KUKA KRL program: MyProgram_024().src

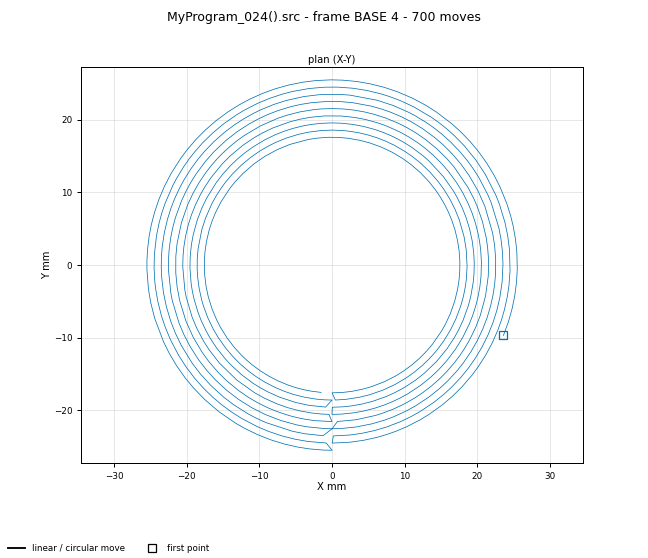
[picture p0: tool path of MyProgram_024().src in frame BASE 4, 700 of 700 moves have a stored position in this frame; points joined in program order, loops and branches not executed]
&ACCESS RVP
&REL 1
&PARAM TEMPLATE = C:\KRC\Roboter\Template\vorgabe
&PARAM EDITMASK = *
DEF MyProgram_024()
; ---- Setting reference (Base) ----
$BASE = BASE_DATA[4]

; --------------------------
; ---- Setting tool (TCP) ----
$TOOL = TOOL_DATA[3]
; --------------------------

$VEL.CP = VEL_APROX_PRINT
Startdeposition()
$VEL.CP = VEL_PRINT
LIN {X 23.5974,Y -9.6926,Z 57,A -28.3314,B 24.8282,C -3.0231,E1 25.1491,E2 -248.9797} C_DIS
LIN {X 24.2747,Y -7.8424,Z 57,A -24.218,B 24.8271,C -3.0328,E1 25.1528,E2 -253.093} C_DIS
LIN {X 24.7886,Y -6.0243,Z 57,A -19.8606,B 24.8255,C -3.0472,E1 25.1559,E2 -257.4593} C_DIS
LIN {X 25.1579,Y -4.2259,Z 57,A -15.7449,B 24.824,C -3.0599,E1 25.158,E2 -261.5811} C_DIS
LIN {X 25.4033,Y -2.3332,Z 57,A -11.6875,B 24.8228,C -3.0706,E1 25.1593,E2 -265.6398} C_DIS
LIN {X 25.5049,Y -0.5316,Z 57,A -6.9801,B 24.8204,C -3.0909,E1 25.1598,E2 -270.3674} C_DIS
LIN {X 25.4452,Y 1.817,Z 57,A -2.3084,B 24.8193,C -3.1002,E1 25.1592,E2 -275.0333} C_DIS
LIN {X 25.2568,Y 3.5873,Z 57,A 1.7378,B 24.8178,C -3.113,E1 25.1578,E2 -279.0859} C_DIS
LIN {X 24.9227,Y 5.4431,Z 57,A 5.9882,B 24.8163,C -3.1259,E1 25.1554,E2 -283.3422} C_DIS
LIN {X 24.5979,Y 6.7615,Z 57,A 9.2535,B 24.8149,C -3.1375,E1 25.1531,E2 -286.6161} C_DIS
LIN {X 24.0961,Y 8.3747,Z 57,A 13.4975,B 24.813,C -3.1536,E1 25.1492,E2 -290.8744} C_DIS
LIN {X 23.1444,Y 10.7284,Z 57,A 18.4456,B 24.8121,C -3.1608,E1 25.1437,E2 -295.8124} C_DIS
LIN {X 22.2888,Y 12.4091,Z 57,A 22.6691,B 24.8108,C -3.1719,E1 25.1382,E2 -300.0401} C_DIS
LIN {X 21.2717,Y 14.0817,Z 57,A 27.0653,B 24.8095,C -3.1829,E1 25.1316,E2 -304.4403} C_DIS
LIN {X 20.123,Y 15.6796,Z 57,A 31.2435,B 24.8085,C -3.1908,E1 25.1246,E2 -308.6172} C_DIS
LIN {X 19.0448,Y 16.9728,Z 57,A 35.1391,B 24.8074,C -3.2004,E1 25.1175,E2 -312.518} C_DIS
LIN {X 17.7974,Y 18.2769,Z 57,A 39.241,B 24.8063,C -3.2093,E1 25.1094,E2 -316.6237} C_DIS
LIN {X 16.5553,Y 19.4087,Z 57,A 43.3186,B 24.805,C -3.2197,E1 25.1008,E2 -320.7097} C_DIS
LIN {X 14.3642,Y 21.082,Z 57,A 49.1701,B 24.8042,C -3.2265,E1 25.0876,E2 -326.5568} C_DIS
LIN {X 12.7921,Y 22.0714,Z 57,A 53.3227,B 24.8035,C -3.2324,E1 25.0777,E2 -330.7103} C_DIS
LIN {X 11.0794,Y 22.9786,Z 57,A 57.9272,B 24.8025,C -3.2401,E1 25.0662,E2 -335.3208} C_DIS
LIN {X 9.0363,Y 23.856,Z 57,A 62.7399,B 24.8021,C -3.2433,E1 25.0537,E2 -340.1302} C_DIS
LIN {X 7.1477,Y 24.4882,Z 57,A 67.1046,B 24.8019,C -3.2456,E1 25.0421,E2 -344.4925} C_DIS
LIN {X 5.2619,Y 24.9618,Z 57,A 71.4856,B 24.8016,C -3.248,E1 25.0302,E2 -348.873} C_DIS
LIN {X 3.3906,Y 25.284,Z 57,A 75.7755,B 24.8014,C -3.2494,E1 25.0184,E2 -353.1622} C_DIS
LIN {X 1.4533,Y 25.4688,Z 57,A 79.6015,B 24.8019,C -3.245,E1 25.0077,E2 -356.9757} C_DIS
LIN {X -0.1497,Y 25.5099,Z 57,A 83.8568,B 24.8013,C -3.2498,E1 24.9958,E2 -361.2422} C_DIS
LIN {X -2.166,Y 25.4178,Z 57,A 88.1783,B 24.8018,C -3.2463,E1 24.9838,E2 -365.5568} C_DIS
LIN {X -3.9428,Y 25.2038,Z 57,A 92.4799,B 24.8018,C -3.246,E1 24.9719,E2 -369.8611} C_DIS
LIN {X -5.9691,Y 24.8019,Z 57,A 96.9208,B 24.8025,C -3.2405,E1 24.9598,E2 -374.2945} C_DIS
LIN {X -7.8398,Y 24.2755,Z 57,A 101.2468,B 24.8031,C -3.2355,E1 24.9483,E2 -378.6158} C_DIS
LIN {X -9.6059,Y 23.6324,Z 57,A 105.5538,B 24.8037,C -3.2306,E1 24.9371,E2 -382.9204} C_DIS
LIN {X -11.3897,Y 22.8266,Z 57,A 109.6739,B 24.8047,C -3.2221,E1 24.9267,E2 -387.0305} C_DIS
LIN {X -12.8693,Y 22.0267,Z 57,A 113.4295,B 24.8055,C -3.2156,E1 24.9175,E2 -390.7813} C_DIS
LIN {X -14.3968,Y 21.0597,Z 57,A 117.8771,B 24.8061,C -3.2105,E1 24.9072,E2 -395.2315} C_DIS
LIN {X -15.9987,Y 19.8702,Z 57,A 122.312,B 24.8073,C -3.201,E1 24.8974,E2 -399.6598} C_DIS
LIN {X -17.4613,Y 18.5978,Z 57,A 126.6023,B 24.8085,C -3.1909,E1 24.8885,E2 -403.9432} C_DIS
LIN {X -18.7226,Y 17.3277,Z 57,A 130.7535,B 24.8096,C -3.1821,E1 24.8805,E2 -408.0912} C_DIS
LIN {X -19.9337,Y 15.9198,Z 57,A 134.7937,B 24.8109,C -3.1708,E1 24.8733,E2 -412.1231} C_DIS
LIN {X -20.8288,Y 14.7286,Z 57,A 138.4822,B 24.8117,C -3.164,E1 24.8673,E2 -415.8132} C_DIS
LIN {X -22.187,Y 12.5909,Z 57,A 144.0705,B 24.8137,C -3.1477,E1 24.8592,E2 -421.3912} C_DIS
LIN {X -23.0971,Y 10.8307,Z 57,A 148.4759,B 24.8152,C -3.1346,E1 24.8538,E2 -425.789} C_DIS
LIN {X -23.8551,Y 9.0389,Z 57,A 152.9416,B 24.8167,C -3.1222,E1 24.8491,E2 -430.25} C_DIS
LIN {X -24.4663,Y 7.2223,Z 57,A 157.3061,B 24.8182,C -3.1095,E1 24.8455,E2 -434.609} C_DIS
LIN {X -24.9012,Y 5.5426,Z 57,A 160.8222,B 24.8199,C -3.0955,E1 24.8432,E2 -438.1121} C_DIS
LIN {X -25.2019,Y 3.9555,Z 57,A 164.8469,B 24.8209,C -3.0864,E1 24.8413,E2 -442.1389} C_DIS
LIN {X -25.4178,Y 2.1663,Z 57,A 168.8418,B 24.8224,C -3.0735,E1 24.8401,E2 -446.1268} C_DIS
LIN {X -25.5037,Y 0.5661,Z 57,A 171.8056,B 24.8241,C -3.0589,E1 24.8398,E2 -449.0735} C_DIS
LIN {X -25.5018,Y -0.6552,Z 57,A 175.5636,B 24.8245,C -3.0558,E1 24.84,E2 -452.8467} C_DIS
LIN {X -25.2925,Y -3.3258,Z 57,A -178.4748,B 24.8266,C -3.037,E1 24.8416,E2 -458.7989} C_DIS
LIN {X -24.9832,Y -5.1588,Z 57,A -174.3635,B 24.8281,C -3.024,E1 24.8438,E2 -462.9035} C_DIS
LIN {X -24.4374,Y -7.3208,Z 57,A -168.6261,B 24.8293,C -3.0134,E1 24.8481,E2 -468.6488} C_DIS
LIN {X -23.2088,Y -10.5894,Z 57,A -161.9405,B 24.8326,C -2.9847,E1 24.855,E2 -475.3029} C_DIS
LIN {X -22.4165,Y -12.1769,Z 57,A -157.4517,B 24.8334,C -2.977,E1 24.8608,E2 -479.7974} C_DIS
LIN {X -21.4191,Y -13.8564,Z 57,A -153.0174,B 24.8347,C -2.9662,E1 24.8673,E2 -484.2283} C_DIS
LIN {X -20.2689,Y -15.4905,Z 57,A -148.5031,B 24.8358,C -2.9557,E1 24.8748,E2 -488.7393} C_DIS
LIN {X -19.0968,Y -16.9142,Z 57,A -144.3818,B 24.8369,C -2.9463,E1 24.8823,E2 -492.857} C_DIS
LIN {X -17.5052,Y -18.5563,Z 57,A -138.9873,B 24.8378,C -2.9376,E1 24.893,E2 -498.2534} C_DIS
LIN {X -15.5207,Y -20.2452,Z 57,A -132.526,B 24.8385,C -2.9313,E1 24.9071,E2 -504.724} C_DIS
LIN {X -13.3044,Y -21.7661,Z 57,A -127.5351,B 24.8404,C -2.9147,E1 24.9187,E2 -509.6914} C_DIS
LIN {X -12.0506,Y -22.4847,Z 57,A -123.9663,B 24.8406,C -2.9128,E1 24.9274,E2 -513.2659} C_DIS
LIN {X -10.2372,Y -23.3661,Z 57,A -119.449,B 24.8411,C -2.9078,E1 24.9389,E2 -517.7823} C_DIS
LIN {X -8.4417,Y -24.0728,Z 57,A -115.0933,B 24.8415,C -2.9042,E1 24.9503,E2 -522.1384} C_DIS
LIN {X -6.6102,Y -24.6387,Z 57,A -110.8019,B 24.8418,C -2.9013,E1 24.9618,E2 -526.4299} C_DIS
LIN {X -4.7543,Y -25.0634,Z 57,A -106.5325,B 24.842,C -2.8994,E1 24.9735,E2 -530.6999} C_DIS
LIN {X -3.1602,Y -25.314,Z 57,A -102.8759,B 24.842,C -2.899,E1 24.9836,E2 -534.3583} C_DIS
LIN {X -1.1779,Y -25.483,Z 57,A -98.4765,B 24.8421,C -2.8985,E1 24.9958,E2 -538.758} C_DIS
LIN {X 0.0017,Y -25.5054,Z 57,A -95.9196,B 24.8421,C -2.8983,E1 25.003,E2 -541.3145} C_DIS
Enddeposition()
LIN {X 0.0017,Y -25.5054,Z 57,A -95.9196,B 24.8421,C -2.8983,E1 25.003,E2 -541.3145} C_DIS
Startdeposition()
$VEL.CP = VEL_PRINT
LIN {X -0.8162,Y -24.5086,Z 57,A -100.4797,B 24.8428,C -2.8929,E1 24.9902,E2 -536.7411} C_DIS
LIN {X -3.343,Y -24.2934,Z 57,A -105.8436,B 24.8422,C -2.898,E1 24.9753,E2 -531.386} C_DIS
LIN {X -5.1134,Y -23.9829,Z 57,A -110.0123,B 24.842,C -2.8998,E1 24.9639,E2 -527.217} C_DIS
LIN {X -6.9312,Y -23.5218,Z 57,A -114.4025,B 24.8417,C -2.9024,E1 24.9521,E2 -522.8262} C_DIS
LIN {X -8.7143,Y -22.9213,Z 57,A -118.9495,B 24.8414,C -2.905,E1 24.9401,E2 -518.2763} C_DIS
LIN {X -10.284,Y -22.2612,Z 57,A -123.2424,B 24.8412,C -2.9071,E1 24.9292,E2 -513.978} C_DIS
LIN {X -12.5044,Y -21.0944,Z 57,A -128.2625,B 24.8397,C -2.9204,E1 24.917,E2 -508.9752} C_DIS
LIN {X -13.8365,Y -20.2452,Z 57,A -132.1033,B 24.8392,C -2.925,E1 24.908,E2 -505.133} C_DIS
LIN {X -15.1839,Y -19.2557,Z 57,A -136.3359,B 24.8387,C -2.9296,E1 24.8986,E2 -500.8961} C_DIS
LIN {X -16.5203,Y -18.1223,Z 57,A -140.2889,B 24.8378,C -2.9382,E1 24.8903,E2 -496.9481} C_DIS
LIN {X -17.6802,Y -16.9922,Z 57,A -144.3432,B 24.8371,C -2.9444,E1 24.8823,E2 -492.8914} C_DIS
LIN {X -18.9103,Y -15.6122,Z 57,A -148.5343,B 24.8359,C -2.9548,E1 24.8747,E2 -488.7059} C_DIS
LIN {X -20.0676,Y -14.0935,Z 57,A -153.0925,B 24.8348,C -2.9648,E1 24.8672,E2 -484.1497} C_DIS
LIN {X -21.1149,Y -12.4698,Z 57,A -158.0469,B 24.8338,C -2.974,E1 24.86,E2 -479.1918} C_DIS
LIN {X -22.2501,Y -10.3079,Z 57,A -162.6904,B 24.8314,C -2.9949,E1 24.8542,E2 -474.5733} C_DIS
LIN {X -22.9755,Y -8.5693,Z 57,A -167.9487,B 24.8305,C -3.0028,E1 24.8487,E2 -469.3047} C_DIS
LIN {X -23.5095,Y -6.9732,Z 57,A -171.3197,B 24.8289,C -3.0171,E1 24.8459,E2 -465.9484} C_DIS
LIN {X -24.0022,Y -5.0236,Z 57,A -177.0526,B 24.8279,C -3.026,E1 24.8423,E2 -460.2034} C_DIS
LIN {X -24.3161,Y -3.1693,Z 57,A 179.493,B 24.8258,C -3.044,E1 24.8409,E2 -456.7713} C_DIS
LIN {X -24.4335,Y -2.0783,Z 57,A 176.5746,B 24.8251,C -3.0501,E1 24.8401,E2 -453.8502} C_DIS
LIN {X -24.5179,Y -0.4555,Z 57,A 172.7447,B 24.8238,C -3.0618,E1 24.8398,E2 -450.0252} C_DIS
LIN {X -24.4799,Y 1.4247,Z 57,A 168.2785,B 24.8222,C -3.0751,E1 24.8403,E2 -445.5641} C_DIS
LIN {X -24.1837,Y 4.0593,Z 57,A 161.6445,B 24.8202,C -3.0923,E1 24.8427,E2 -438.9316} C_DIS
LIN {X -23.8193,Y 5.828,Z 57,A 158.2213,B 24.8183,C -3.1091,E1 24.8448,E2 -435.5285} C_DIS
LIN {X -23.4594,Y 7.1394,Z 57,A 154.6095,B 24.8174,C -3.1167,E1 24.8476,E2 -431.914} C_DIS
LIN {X -23.0092,Y 8.4797,Z 57,A 150.6203,B 24.8166,C -3.1233,E1 24.8514,E2 -427.918} C_DIS
LIN {X -21.9422,Y 10.9487,Z 57,A 145.374,B 24.8138,C -3.1467,E1 24.8575,E2 -422.6991} C_DIS
LIN {X -21.429,Y 11.9218,Z 57,A 142.3229,B 24.8132,C -3.1515,E1 24.8616,E2 -419.6435} C_DIS
LIN {X -20.4509,Y 13.5307,Z 57,A 138.2469,B 24.8116,C -3.1652,E1 24.8676,E2 -415.5796} C_DIS
LIN {X -19.6571,Y 14.6605,Z 57,A 135.1759,B 24.8105,C -3.1745,E1 24.8726,E2 -412.516} C_DIS
LIN {X -18.9586,Y 15.5535,Z 57,A 132.147,B 24.8099,C -3.1793,E1 24.8779,E2 -409.4842} C_DIS
LIN {X -17.8107,Y 16.8557,Z 57,A 127.8837,B 24.8089,C -3.188,E1 24.886,E2 -405.2229} C_DIS
LIN {X -16.3984,Y 18.2327,Z 57,A 123.2379,B 24.8076,C -3.1982,E1 24.8954,E2 -400.5827} C_DIS
LIN {X -14.9317,Y 19.4519,Z 57,A 118.4259,B 24.8068,C -3.2055,E1 24.9059,E2 -395.7702} C_DIS
LIN {X -13.2236,Y 20.6511,Z 57,A 114.2463,B 24.8051,C -3.2189,E1 24.9156,E2 -391.6087} C_DIS
LIN {X -12.1128,Y 21.3219,Z 57,A 110.8599,B 24.8048,C -3.222,E1 24.9237,E2 -388.2195} C_DIS
LIN {X -10.3297,Y 22.24,Z 57,A 106.1341,B 24.8039,C -3.229,E1 24.9356,E2 -383.498} C_DIS
LIN {X -8.5761,Y 22.9732,Z 57,A 101.6704,B 24.8032,C -3.2347,E1 24.9472,E2 -379.0384} C_DIS
LIN {X -6.7424,Y 23.5769,Z 57,A 97.607,B 24.8022,C -3.2427,E1 24.958,E2 -374.9871} C_DIS
LIN {X -5.4397,Y 23.9109,Z 57,A 93.8987,B 24.8023,C -3.2417,E1 24.968,E2 -371.2712} C_DIS
LIN {X -3.1801,Y 24.3149,Z 57,A 88.636,B 24.8018,C -3.246,E1 24.9825,E2 -366.0141} C_DIS
LIN {X -1.0603,Y 24.4985,Z 57,A 83.951,B 24.8013,C -3.2502,E1 24.9956,E2 -361.3373} C_DIS
LIN {X 0.7326,Y 24.5108,Z 57,A 79.1328,B 24.8018,C -3.246,E1 25.009,E2 -356.5096} C_DIS
LIN {X 2.8302,Y 24.3581,Z 57,A 74.5816,B 24.8015,C -3.2484,E1 25.0217,E2 -351.9668} C_DIS
LIN {X 4.7024,Y 24.067,Z 57,A 69.4413,B 24.8024,C -3.2409,E1 25.0358,E2 -346.8144} C_DIS
LIN {X 6.6864,Y 23.5927,Z 57,A 65.7695,B 24.8017,C -3.2473,E1 25.0457,E2 -343.1636} C_DIS
LIN {X 7.8457,Y 23.2327,Z 57,A 62.9862,B 24.8019,C -3.2456,E1 25.0531,E2 -340.3814} C_DIS
LIN {X 9.3946,Y 22.6509,Z 57,A 58.3374,B 24.8032,C -3.2349,E1 25.0652,E2 -335.7176} C_DIS
LIN {X 11.2204,Y 21.8043,Z 57,A 53.3946,B 24.8041,C -3.2271,E1 25.0775,E2 -330.7694} C_DIS
LIN {X 13.6548,Y 20.3686,Z 57,A 47.7894,B 24.8041,C -3.2267,E1 25.0908,E2 -325.1811} C_DIS
LIN {X 14.7224,Y 19.6108,Z 57,A 44.6371,B 24.8049,C -3.2207,E1 25.0979,E2 -322.0257} C_DIS
LIN {X 15.8085,Y 18.7463,Z 57,A 41.3255,B 24.8057,C -3.2141,E1 25.1051,E2 -318.7111} C_DIS
LIN {X 16.8223,Y 17.8422,Z 57,A 37.9278,B 24.8067,C -3.2056,E1 25.1121,E2 -315.3071} C_DIS
LIN {X 18.1912,Y 16.4443,Z 57,A 33.2587,B 24.808,C -3.1949,E1 25.121,E2 -310.6329} C_DIS
LIN {X 19.8061,Y 14.4585,Z 57,A 26.7554,B 24.8104,C -3.1756,E1 25.1321,E2 -304.1145} C_DIS
LIN {X 21.0994,Y 12.4958,Z 57,A 21.1531,B 24.8122,C -3.1604,E1 25.1403,E2 -298.5048} C_DIS
LIN {X 22.5618,Y 9.6075,Z 57,A 15.2266,B 24.8125,C -3.1574,E1 25.1474,E2 -292.6028} C_DIS
LIN {X 23.0349,Y 8.4095,Z 57,A 11.0682,B 24.815,C -3.1364,E1 25.1515,E2 -288.4179} C_DIS
LIN {X 23.8129,Y 5.8544,Z 57,A 5.2905,B 24.8166,C -3.123,E1 25.1559,E2 -282.6417} C_DIS
LIN {X 24.1913,Y 4.0145,Z 57,A 0.9918,B 24.8181,C -3.1108,E1 25.1581,E2 -278.339} C_DIS
LIN {X 24.4273,Y 2.1521,Z 57,A -4.0505,B 24.8205,C -3.09,E1 25.1595,E2 -273.2775} C_DIS
LIN {X 24.5108,Y -0.7385,Z 57,A -10.2973,B 24.8223,C -3.0746,E1 25.1595,E2 -267.0314} C_DIS
LIN {X 24.3597,Y -2.8172,Z 57,A -14.5236,B 24.8232,C -3.0666,E1 25.1585,E2 -262.8111} C_DIS
LIN {X 24.1391,Y -4.317,Z 57,A -18.4922,B 24.825,C -3.0508,E1 25.1567,E2 -258.8285} C_DIS
LIN {X 23.7335,Y -6.1692,Z 57,A -22.9517,B 24.8266,C -3.0368,E1 25.1538,E2 -254.3617} C_DIS
LIN {X 23.2874,Y -7.6821,Z 57,A -26.0063,B 24.8271,C -3.0326,E1 25.1513,E2 -251.3144} C_DIS
LIN {X 22.8272,Y -8.9576,Z 57,A -29.674,B 24.8288,C -3.0176,E1 25.1477,E2 -247.6317} C_DIS
LIN {X 22.0848,Y -10.6578,Z 57,A -33.9482,B 24.8302,C -3.0056,E1 25.1427,E2 -243.3521} C_DIS
LIN {X 21.2084,Y -12.3104,Z 57,A -38.7058,B 24.8321,C -2.9891,E1 25.1362,E2 -238.5801} C_DIS
LIN {X 20.088,Y -14.0645,Z 57,A -42.8035,B 24.8326,C -2.9841,E1 25.1299,E2 -234.4909} C_DIS
LIN {X 19.2809,Y -15.152,Z 57,A -46.285,B 24.834,C -2.9724,E1 25.1239,E2 -230.9983} C_DIS
LIN {X 17.9089,Y -16.7511,Z 57,A -51.0916,B 24.8352,C -2.9614,E1 25.115,E2 -226.1872} C_DIS
LIN {X 16.5964,Y -18.0525,Z 57,A -55.5524,B 24.8365,C -2.95,E1 25.106,E2 -221.7177} C_DIS
LIN {X 15.203,Y -19.2406,Z 57,A -60.0611,B 24.8377,C -2.9385,E1 25.0962,E2 -217.1988} C_DIS
LIN {X 13.3435,Y -20.5736,Z 57,A -64.6446,B 24.8381,C -2.9356,E1 25.0857,E2 -212.6241} C_DIS
LIN {X 12.0817,Y -21.3389,Z 57,A -68.6968,B 24.8394,C -2.9236,E1 25.0759,E2 -208.5558} C_DIS
LIN {X 10.2776,Y -22.2641,Z 57,A -73.2647,B 24.84,C -2.9178,E1 25.0644,E2 -203.9862} C_DIS
LIN {X 8.8215,Y -22.8801,Z 57,A -76.4646,B 24.84,C -2.9173,E1 25.0562,E2 -200.7925} C_DIS
LIN {X 7.6695,Y -23.2913,Z 57,A -79.7044,B 24.8408,C -2.9103,E1 25.0476,E2 -197.5423} C_DIS
LIN {X 6.2074,Y -23.7233,Z 57,A -83.3054,B 24.8413,C -2.9062,E1 25.0379,E2 -193.9375} C_DIS
LIN {X 4.3572,Y -24.1319,Z 57,A -87.7631,B 24.8417,C -2.9022,E1 25.0257,E2 -189.4757} C_DIS
LIN {X 2.4426,Y -24.4001,Z 57,A -92.708,B 24.8424,C -2.8959,E1 25.0119,E2 -184.5194} C_DIS
LIN {X 0.0065,Y -24.5225,Z 57,A -95.59,B 24.84,C -2.9177,E1 25.004,E2 -181.6903} C_DIS
Enddeposition()
LIN {X 0.0065,Y -24.5225,Z 57,A -95.59,B 24.84,C -2.9177,E1 25.004,E2 -181.6903} C_DIS
Startdeposition()
$VEL.CP = VEL_PRINT
LIN {X 0.1728,Y -23.5332,Z 57,A -95.0814,B 24.8381,C -2.9354,E1 25.0056,E2 -182.241} C_DIS
LIN {X 2.4377,Y -23.4068,Z 57,A -90.2543,B 24.8384,C -2.9321,E1 25.019,E2 -187.0578} C_DIS
LIN {X 4.046,Y -23.1837,Z 57,A -85.8902,B 24.8377,C -2.9385,E1 25.031,E2 -191.4327} C_DIS
LIN {X 5.8549,Y -22.7937,Z 57,A -81.6004,B 24.8375,C -2.9408,E1 25.0427,E2 -195.722} C_DIS
LIN {X 7.5378,Y -22.2935,Z 57,A -76.8383,B 24.8364,C -2.9502,E1 25.0554,E2 -200.4977} C_DIS
LIN {X 9.3798,Y -21.5835,Z 57,A -72.4094,B 24.8361,C -2.9534,E1 25.0668,E2 -204.9239} C_DIS
LIN {X 10.8597,Y -20.8786,Z 57,A -68.6996,B 24.8357,C -2.9571,E1 25.0761,E2 -208.6324} C_DIS
LIN {X 12.1662,Y -20.1452,Z 57,A -64.7539,B 24.8346,C -2.9664,E1 25.0856,E2 -212.5883} C_DIS
LIN {X 14.0298,Y -18.8948,Z 57,A -59.3169,B 24.8334,C -2.9769,E1 25.0981,E2 -218.0315} C_DIS
LIN {X 15.404,Y -17.7921,Z 57,A -55.2869,B 24.8327,C -2.9836,E1 25.1067,E2 -222.0618} C_DIS
LIN {X 16.512,Y -16.7688,Z 57,A -51.5293,B 24.8316,C -2.993,E1 25.1143,E2 -225.8261} C_DIS
LIN {X 17.7863,Y -15.411,Z 57,A -47.3126,B 24.8308,C -3.0008,E1 25.1222,E2 -230.0428} C_DIS
LIN {X 18.8448,Y -14.0963,Z 57,A -42.8149,B 24.8291,C -3.0156,E1 25.13,E2 -234.5542} C_DIS
LIN {X 19.7762,Y -12.757,Z 57,A -39.0539,B 24.8281,C -3.0241,E1 25.1358,E2 -238.3168} C_DIS
LIN {X 20.6346,Y -11.3168,Z 57,A -34.7573,B 24.8265,C -3.0379,E1 25.1418,E2 -242.6239} C_DIS
LIN {X 21.4569,Y -9.666,Z 57,A -30.3654,B 24.8251,C -3.0499,E1 25.147,E2 -247.0205} C_DIS
LIN {X 22.1456,Y -7.9621,Z 57,A -25.9982,B 24.8237,C -3.0621,E1 25.1514,E2 -251.3923} C_DIS
LIN {X 22.6902,Y -6.2446,Z 57,A -21.4937,B 24.822,C -3.0768,E1 25.1549,E2 -255.9059} C_DIS
LIN {X 23.0932,Y -4.5333,Z 57,A -17.297,B 24.8206,C -3.0891,E1 25.1574,E2 -260.1073} C_DIS
LIN {X 23.4185,Y -2.3263,Z 57,A -11.3589,B 24.818,C -3.1117,E1 25.1594,E2 -266.0637} C_DIS
LIN {X 23.5357,Y 0.142,Z 57,A -5.7796,B 24.8163,C -3.1255,E1 25.1597,E2 -271.6427} C_DIS
LIN {X 23.461,Y 1.8498,Z 57,A -2.1065,B 24.8154,C -3.1331,E1 25.1591,E2 -275.3119} C_DIS
LIN {X 23.2709,Y 3.509,Z 57,A 2.26,B 24.8136,C -3.1488,E1 25.1575,E2 -279.6899} C_DIS
LIN {X 22.9699,Y 5.1217,Z 57,A 7.3044,B 24.8108,C -3.1723,E1 25.1545,E2 -284.7608} C_DIS
LIN {X 21.9227,Y 8.557,Z 57,A 14.7705,B 24.8094,C -3.1836,E1 25.1478,E2 -292.2114} C_DIS
LIN {X 21.4484,Y 9.6849,Z 57,A 18.4083,B 24.8076,C -3.1989,E1 25.1437,E2 -295.8657} C_DIS
LIN {X 20.1752,Y 12.1166,Z 57,A 24.0792,B 24.8067,C -3.2057,E1 25.136,E2 -301.5232} C_DIS
LIN {X 19.342,Y 13.4062,Z 57,A 27.7241,B 24.8057,C -3.2141,E1 25.1304,E2 -305.1698} C_DIS
LIN {X 18.6123,Y 14.4023,Z 57,A 30.9154,B 24.8046,C -3.2231,E1 25.125,E2 -308.3672} C_DIS
LIN {X 17.7311,Y 15.4742,Z 57,A 34.6473,B 24.8033,C -3.2342,E1 25.1183,E2 -312.1085} C_DIS
LIN {X 16.411,Y 16.8681,Z 57,A 39.2881,B 24.8021,C -3.2436,E1 25.1091,E2 -316.7517} C_DIS
LIN {X 15.0831,Y 18.0649,Z 57,A 43.2663,B 24.8016,C -3.2481,E1 25.1008,E2 -320.7252} C_DIS
LIN {X 13.9703,Y 18.9386,Z 57,A 46.6692,B 24.8009,C -3.2537,E1 25.0932,E2 -324.1289} C_DIS
LIN {X 12.9444,Y 19.6541,Z 57,A 49.9429,B 24.8,C -3.2607,E1 25.0856,E2 -327.4081} C_DIS
LIN {X 11.4624,Y 20.5535,Z 57,A 53.7393,B 24.7998,C -3.2627,E1 25.0765,E2 -331.1978} C_DIS
LIN {X 10.4876,Y 21.0677,Z 57,A 56.7363,B 24.799,C -3.2688,E1 25.069,E2 -334.2013} C_DIS
LIN {X 8.401,Y 21.9831,Z 57,A 63.2209,B 24.7973,C -3.2827,E1 25.0522,E2 -340.7039} C_DIS
LIN {X 6.1651,Y 22.7118,Z 57,A 69.2316,B 24.7965,C -3.289,E1 25.0361,E2 -346.7194} C_DIS
LIN {X 2.4387,Y 23.407,Z 57,A 76.8785,B 24.7978,C -3.2788,E1 25.0151,E2 -354.3345} C_DIS
LIN {X 0.9169,Y 23.5157,Z 57,A 81.442,B 24.797,C -3.2853,E1 25.0023,E2 -358.9119} C_DIS
LIN {X -1.7418,Y 23.469,Z 57,A 88.3308,B 24.7969,C -3.2862,E1 24.9831,E2 -365.8046} C_DIS
LIN {X -3.8729,Y 23.213,Z 57,A 93.2665,B 24.7975,C -3.2807,E1 24.9695,E2 -370.7313} C_DIS
LIN {X -6.3555,Y 22.6591,Z 57,A 98.872,B 24.7988,C -3.2708,E1 24.9544,E2 -376.3211} C_DIS
LIN {X -8.0275,Y 22.1221,Z 57,A 103.6927,B 24.7989,C -3.2693,E1 24.9416,E2 -381.1476} C_DIS
LIN {X -9.8388,Y 21.3783,Z 57,A 107.5208,B 24.8005,C -3.2566,E1 24.9319,E2 -384.9542} C_DIS
LIN {X -10.8189,Y 20.8996,Z 57,A 110.3642,B 24.8009,C -3.2536,E1 24.9248,E2 -387.798} C_DIS
LIN {X -12.1998,Y 20.1248,Z 57,A 114.7094,B 24.8013,C -3.2499,E1 24.9143,E2 -392.1474} C_DIS
LIN {X -13.5599,Y 19.2346,Z 57,A 118.3647,B 24.8025,C -3.2405,E1 24.9059,E2 -395.7926} C_DIS
LIN {X -14.8546,Y 18.2533,Z 57,A 122.6984,B 24.8032,C -3.2345,E1 24.8964,E2 -400.1278} C_DIS
LIN {X -16.2922,Y 16.9825,Z 57,A 127.248,B 24.8046,C -3.2233,E1 24.8871,E2 -404.6691} C_DIS
LIN {X -17.5749,Y 15.6515,Z 57,A 131.1506,B 24.8063,C -3.2093,E1 24.8796,E2 -408.5551} C_DIS
LIN {X -18.4413,Y 14.6201,Z 57,A 134.8568,B 24.807,C -3.2032,E1 24.8731,E2 -412.264} C_DIS
LIN {X -19.46,Y 13.2342,Z 57,A 139.5696,B 24.808,C -3.1948,E1 24.8655,E2 -416.9797} C_DIS
LIN {X -20.3847,Y 11.7603,Z 57,A 143.344,B 24.8097,C -3.1807,E1 24.8601,E2 -420.74} C_DIS
LIN {X -21.0589,Y 10.5045,Z 57,A 146.9565,B 24.8108,C -3.1715,E1 24.8555,E2 -424.3497} C_DIS
LIN {X -21.704,Y 9.0975,Z 57,A 150.5983,B 24.8122,C -3.1599,E1 24.8514,E2 -427.9837} C_DIS
LIN {X -22.1837,Y 7.8563,Z 57,A 153.7951,B 24.8134,C -3.15,E1 24.8483,E2 -431.1748} C_DIS
LIN {X -22.6616,Y 6.3466,Z 57,A 158,B 24.8146,C -3.14,E1 24.8449,E2 -435.3799} C_DIS
LIN {X -23.1003,Y 4.4958,Z 57,A 162.871,B 24.8162,C -3.1268,E1 24.8421,E2 -440.2481} C_DIS
LIN {X -23.3938,Y 2.5612,Z 57,A 167.5401,B 24.818,C -3.1116,E1 24.8404,E2 -444.9086} C_DIS
LIN {X -23.5009,Y 1.2387,Z 57,A 170.6619,B 24.8192,C -3.101,E1 24.8399,E2 -448.0237} C_DIS
LIN {X -23.5327,Y -0.2865,Z 57,A 174.6171,B 24.8204,C -3.0906,E1 24.8399,E2 -451.9778} C_DIS
LIN {X -23.4759,Y -1.6466,Z 57,A 178.1601,B 24.8215,C -3.0814,E1 24.8405,E2 -455.5202} C_DIS
LIN {X -23.2265,Y -3.7916,Z 57,A -176.8014,B 24.8235,C -3.0643,E1 24.8425,E2 -460.5478} C_DIS
LIN {X -22.8332,Y -5.6983,Z 57,A -171.9567,B 24.8251,C -3.0507,E1 24.8455,E2 -465.3883} C_DIS
LIN {X -22.2244,Y -7.7396,Z 57,A -167.2191,B 24.827,C -3.0334,E1 24.8495,E2 -470.1117} C_DIS
LIN {X -21.594,Y -9.3556,Z 57,A -163.471,B 24.8287,C -3.0192,E1 24.8534,E2 -473.8466} C_DIS
LIN {X -20.7533,Y -11.0975,Z 57,A -156.7949,B 24.8289,C -3.0168,E1 24.8619,E2 -480.5529} C_DIS
LIN {X -19.2949,Y -13.4741,Z 57,A -150.9981,B 24.8315,C -2.9945,E1 24.8707,E2 -486.3254} C_DIS
LIN {X -18.1375,Y -14.9959,Z 57,A -146.6587,B 24.8329,C -2.982,E1 24.8782,E2 -490.6553} C_DIS
LIN {X -16.6819,Y -16.6001,Z 57,A -140.4619,B 24.8335,C -2.9763,E1 24.8901,E2 -496.8653} C_DIS
LIN {X -14.9399,Y -18.1837,Z 57,A -136.0488,B 24.8356,C -2.9576,E1 24.8993,E2 -501.251} C_DIS
LIN {X -13.5966,Y -19.2087,Z 57,A -130.4167,B 24.8353,C -2.9602,E1 24.9121,E2 -506.9094} C_DIS
LIN {X -11.5846,Y -20.4852,Z 57,A -126.0331,B 24.8373,C -2.9427,E1 24.9225,E2 -511.2648} C_DIS
LIN {X -10.6358,Y -20.9932,Z 57,A -122.909,B 24.8373,C -2.9428,E1 24.9302,E2 -514.3976} C_DIS
LIN {X -9.1394,Y -21.6865,Z 57,A -117.5528,B 24.8367,C -2.9481,E1 24.9441,E2 -519.7788} C_DIS
LIN {X -5.4206,Y -22.9011,Z 57,A -108.8189,B 24.838,C -2.936,E1 24.9674,E2 -528.4981} C_DIS
LIN {X -3.7056,Y -23.2403,Z 57,A -104.323,B 24.838,C -2.9366,E1 24.9798,E2 -532.9997} C_DIS
LIN {X -1.2416,Y -23.5006,Z 57,A -98.6896,B 24.8383,C -2.9333,E1 24.9955,E2 -538.6277} C_DIS
LIN {X -1.2416,Y -23.5006,Z 57,A -98.6896,B 24.8383,C -2.9333,E1 24.9955,E2 -538.6277} C_DIS
Enddeposition()
LIN {X 0.0024,Y -22.5443,Z 57,A -96.7475,B 24.8373,C -2.9421,E1 25.0009,E2 -540.591} C_DIS
Startdeposition()
$VEL.CP = VEL_PRINT
LIN {X -1.0975,Y -22.5186,Z 57,A -101.3568,B 24.8389,C -2.9282,E1 24.988,E2 -535.9477} C_DIS
LIN {X -3.5647,Y -22.2623,Z 57,A -107.4081,B 24.8386,C -2.9311,E1 24.9712,E2 -529.8989} C_DIS
LIN {X -4.8292,Y -22.0222,Z 57,A -110.4489,B 24.8382,C -2.9341,E1 24.963,E2 -526.8615} C_DIS
LIN {X -7.0619,Y -21.4108,Z 57,A -116.9864,B 24.8382,C -2.9338,E1 24.9454,E2 -520.3122} C_DIS
LIN {X -9.1519,Y -20.6043,Z 57,A -122.2067,B 24.8373,C -2.9424,E1 24.932,E2 -515.1006} C_DIS
LIN {X -11.0272,Y -19.6649,Z 57,A -127.2127,B 24.8363,C -2.951,E1 24.9197,E2 -510.1013} C_DIS
LIN {X -12.8786,Y -18.5053,Z 57,A -133.5973,B 24.8359,C -2.9547,E1 24.9048,E2 -503.7046} C_DIS
LIN {X -14.5308,Y -17.2386,Z 57,A -137.9955,B 24.8343,C -2.969,E1 24.8952,E2 -499.3242} C_DIS
LIN {X -15.9802,Y -15.9041,Z 57,A -144.0867,B 24.8339,C -2.9733,E1 24.883,E2 -493.2181} C_DIS
LIN {X -17.2513,Y -14.5156,Z 57,A -148.173,B 24.8323,C -2.9874,E1 24.8755,E2 -489.1469} C_DIS
LIN {X -18.3805,Y -13.0562,Z 57,A -153.083,B 24.8311,C -2.9974,E1 24.8673,E2 -484.2372} C_DIS
LIN {X -19.613,Y -11.1187,Z 57,A -158.7859,B 24.8294,C -3.0129,E1 24.8591,E2 -478.5421} C_DIS
LIN {X -20.3769,Y -9.6473,Z 57,A -162.9916,B 24.8281,C -3.0243,E1 24.8539,E2 -474.341} C_DIS
LIN {X -21.0959,Y -7.9532,Z 57,A -168.5639,B 24.827,C -3.0336,E1 24.8482,E2 -468.7597} C_DIS
LIN {X -21.9918,Y -4.9646,Z 57,A -175.1454,B 24.8237,C -3.0627,E1 24.8434,E2 -462.2098} C_DIS
LIN {X -22.1902,Y -3.9877,Z 57,A -179.0909,B 24.8235,C -3.0644,E1 24.8414,E2 -458.245} C_DIS
LIN {X -22.5341,Y -0.7175,Z 57,A 173.962,B 24.8198,C -3.096,E1 24.8398,E2 -451.3319} C_DIS
LIN {X -22.5343,Y 0.7109,Z 57,A 169.8955,B 24.8187,C -3.1055,E1 24.84,E2 -447.2636} C_DIS
LIN {X -22.4471,Y 2.1021,Z 57,A 166.4498,B 24.8173,C -3.117,E1 24.8407,E2 -443.8246} C_DIS
LIN {X -22.2387,Y 3.7073,Z 57,A 161.8648,B 24.8161,C -3.1278,E1 24.8426,E2 -439.2383} C_DIS
LIN {X -21.9566,Y 5.1198,Z 57,A 158.7163,B 24.8145,C -3.1412,E1 24.8444,E2 -436.1033} C_DIS
LIN {X -21.5853,Y 6.509,Z 57,A 154.3439,B 24.8135,C -3.1493,E1 24.8478,E2 -431.7251} C_DIS
LIN {X -20.7379,Y 8.8456,Z 57,A 148.27,B 24.8111,C -3.1691,E1 24.8539,E2 -425.6646} C_DIS
LIN {X -20.1229,Y 10.1665,Z 57,A 144.8851,B 24.8097,C -3.1812,E1 24.858,E2 -422.2903} C_DIS
LIN {X -19.4938,Y 11.3272,Z 57,A 141.5426,B 24.8085,C -3.1907,E1 24.8626,E2 -418.9529} C_DIS
LIN {X -18.7266,Y 12.5546,Z 57,A 137.3125,B 24.8076,C -3.1982,E1 24.869,E2 -414.7196} C_DIS
LIN {X -17.426,Y 14.3054,Z 57,A 131.496,B 24.8061,C -3.2112,E1 24.879,E2 -408.9067} C_DIS
LIN {X -16.2599,Y 15.6179,Z 57,A 126.7726,B 24.8049,C -3.2207,E1 24.888,E2 -404.1853} C_DIS
LIN {X -14.6414,Y 17.1446,Z 57,A 121.703,B 24.803,C -3.2361,E1 24.8985,E2 -399.1325} C_DIS
LIN {X -13.1259,Y 18.3307,Z 57,A 117.3753,B 24.8015,C -3.249,E1 24.9081,E2 -394.82} C_DIS
LIN {X -11.5883,Y 19.3393,Z 57,A 111.8006,B 24.801,C -3.2527,E1 24.9213,E2 -389.2363} C_DIS
LIN {X -10.1296,Y 20.1421,Z 57,A 108.1819,B 24.7997,C -3.2629,E1 24.9302,E2 -385.6321} C_DIS
LIN {X -8.9118,Y 20.7092,Z 57,A 104.6157,B 24.7992,C -3.267,E1 24.9393,E2 -382.067} C_DIS
LIN {X -7.4245,Y 21.2877,Z 57,A 100.2934,B 24.7988,C -3.2705,E1 24.9506,E2 -377.7443} C_DIS
LIN {X -5.663,Y 21.8227,Z 57,A 95.9068,B 24.798,C -3.2771,E1 24.9623,E2 -373.3665} C_DIS
LIN {X -4.3288,Y 22.1259,Z 57,A 92.3343,B 24.7977,C -3.2794,E1 24.9721,E2 -369.7951} C_DIS
LIN {X -2.8018,Y 22.3705,Z 57,A 87.8981,B 24.7978,C -3.2785,E1 24.9844,E2 -365.3533} C_DIS
LIN {X -0.6499,Y 22.536,Z 57,A 82.8734,B 24.7972,C -3.2837,E1 24.9983,E2 -360.3394} C_DIS
LIN {X 1.0225,Y 22.5219,Z 57,A 78.4626,B 24.7972,C -3.283,E1 25.0107,E2 -355.9279} C_DIS
LIN {X 2.7642,Y 22.3756,Z 57,A 73.5131,B 24.7978,C -3.2786,E1 25.0244,E2 -350.9714} C_DIS
LIN {X 5.3449,Y 21.9027,Z 57,A 67.4167,B 24.7976,C -3.2801,E1 25.041,E2 -344.886} C_DIS
LIN {X 6.6795,Y 21.5331,Z 57,A 64.3724,B 24.7974,C -3.2814,E1 25.0492,E2 -341.8501} C_DIS
LIN {X 8.101,Y 21.0397,Z 57,A 59.8876,B 24.7985,C -3.2727,E1 25.061,E2 -337.3539} C_DIS
LIN {X 9.5918,Y 20.4036,Z 57,A 56.2634,B 24.7985,C -3.2723,E1 25.0702,E2 -333.7377} C_DIS
LIN {X 10.9079,Y 19.7313,Z 57,A 52.1241,B 24.7996,C -3.2642,E1 25.0804,E2 -329.5908} C_DIS
LIN {X 12.4313,Y 18.8087,Z 57,A 47.2981,B 24.8007,C -3.2547,E1 25.0918,E2 -324.758} C_DIS
LIN {X 14.1128,Y 17.5825,Z 57,A 42.8399,B 24.8009,C -3.2531,E1 25.1017,E2 -320.3121} C_DIS
LIN {X 15.2262,Y 16.6273,Z 57,A 38.644,B 24.8024,C -3.2416,E1 25.1105,E2 -316.1057} C_DIS
LIN {X 16.5615,Y 15.2979,Z 57,A 33.8496,B 24.8036,C -3.2315,E1 25.1198,E2 -311.3079} C_DIS
LIN {X 17.7312,Y 13.9243,Z 57,A 29.7261,B 24.8043,C -3.2255,E1 25.1271,E2 -307.1892} C_DIS
LIN {X 18.8636,Y 12.347,Z 57,A 24.2105,B 24.8065,C -3.2078,E1 25.1358,E2 -301.6587} C_DIS
LIN {X 20.0916,Y 10.2281,Z 57,A 17.4427,B 24.8091,C -3.186,E1 25.1448,E2 -294.8747} C_DIS
LIN {X 21.0438,Y 8.0902,Z 57,A 11.1548,B 24.8115,C -3.1659,E1 25.1514,E2 -288.5739} C_DIS
LIN {X 22.1049,Y 4.436,Z 57,A 3.275,B 24.8127,C -3.1556,E1 25.157,E2 -280.7151} C_DIS
LIN {X 22.3786,Y 2.7376,Z 57,A -1.8596,B 24.8153,C -3.1344,E1 25.159,E2 -275.5605} C_DIS
LIN {X 22.5299,Y 0.8342,Z 57,A -6.0878,B 24.8163,C -3.1259,E1 25.1597,E2 -271.3371} C_DIS
LIN {X 22.5157,Y -1.1536,Z 57,A -11.3794,B 24.8184,C -3.1076,E1 25.1594,E2 -266.0338} C_DIS
LIN {X 22.3915,Y -2.6304,Z 57,A -14.9457,B 24.8196,C -3.0979,E1 25.1584,E2 -262.4657} C_DIS
LIN {X 22.1763,Y -4.0647,Z 57,A -18.6376,B 24.8209,C -3.0864,E1 25.1567,E2 -258.7682} C_DIS
LIN {X 21.8377,Y -5.6042,Z 57,A -22.6277,B 24.8223,C -3.0742,E1 25.1541,E2 -254.7724} C_DIS
LIN {X 21.3707,Y -7.1821,Z 57,A -26.8978,B 24.8239,C -3.0606,E1 25.1505,E2 -250.4943} C_DIS
LIN {X 20.7335,Y -8.8559,Z 57,A -31.7415,B 24.8258,C -3.0441,E1 25.1454,E2 -245.6381} C_DIS
LIN {X 20.006,Y -10.3957,Z 57,A -35.7287,B 24.8268,C -3.0351,E1 25.1405,E2 -241.6509} C_DIS
LIN {X 19.1355,Y -11.922,Z 57,A -40.1167,B 24.8282,C -3.0234,E1 25.1342,E2 -237.2576} C_DIS
LIN {X 18.1014,Y -13.4398,Z 57,A -45.2455,B 24.8301,C -3.0064,E1 25.1259,E2 -232.1135} C_DIS
LIN {X 17.1837,Y -14.5955,Z 57,A -48.4206,B 24.8306,C -3.0025,E1 25.1202,E2 -228.9438} C_DIS
LIN {X 15.8959,Y -15.9881,Z 57,A -53.2362,B 24.8319,C -2.9909,E1 25.1109,E2 -224.1216} C_DIS
LIN {X 14.7515,Y -17.0493,Z 57,A -57.4269,B 24.8331,C -2.9799,E1 25.1022,E2 -219.9215} C_DIS
LIN {X 13.3291,Y -18.1834,Z 57,A -62.3176,B 24.8345,C -2.9678,E1 25.0913,E2 -215.0199} C_DIS
LIN {X 11.4809,Y -19.4035,Z 57,A -67.3653,B 24.835,C -2.9628,E1 25.0794,E2 -209.9764} C_DIS
LIN {X 10.1002,Y -20.1567,Z 57,A -71.0613,B 24.8355,C -2.9589,E1 25.0702,E2 -206.2815} C_DIS
LIN {X 8.399,Y -20.9224,Z 57,A -76.3793,B 24.8368,C -2.947,E1 25.0566,E2 -200.9479} C_DIS
LIN {X 7.228,Y -21.3555,Z 57,A -79.463,B 24.8371,C -2.9438,E1 25.0484,E2 -197.8629} C_DIS
LIN {X 5.4671,Y -21.8725,Z 57,A -84.6564,B 24.8382,C -2.9346,E1 25.0344,E2 -192.6559} C_DIS
LIN {X 3.2443,Y -22.3111,Z 57,A -89.9743,B 24.8382,C -2.9339,E1 25.0198,E2 -187.3418} C_DIS
LIN {X 1.1512,Y -22.5157,Z 57,A -95.0343,B 24.8382,C -2.9336,E1 25.0057,E2 -182.2836} C_DIS
LIN {X 0.0024,Y -22.5443,Z 57,A -96.7474,B 24.8373,C -2.9421,E1 25.0009,E2 -180.591} C_DIS
Enddeposition()
LIN {X 0.0024,Y -22.5443,Z 57,A -96.7474,B 24.8373,C -2.9421,E1 25.0009,E2 -180.591} C_DIS
Startdeposition()
$VEL.CP = VEL_PRINT
LIN {X 0.7335,Y -21.5448,Z 57,A -93.3683,B 24.8341,C -2.9707,E1 25.0106,E2 -184.0372} C_DIS
LIN {X 3.2857,Y -21.3055,Z 57,A -86.369,B 24.8335,C -2.9763,E1 25.03,E2 -191.0445} C_DIS
LIN {X 5.9549,Y -20.7181,Z 57,A -80.7984,B 24.8343,C -2.9693,E1 25.045,E2 -196.5904} C_DIS
LIN {X 7.04,Y -20.375,Z 57,A -76.9146,B 24.8331,C -2.9801,E1 25.0554,E2 -200.4925} C_DIS
LIN {X 8.4969,Y -19.812,Z 57,A -72.8051,B 24.8325,C -2.9855,E1 25.066,E2 -204.6055} C_DIS
LIN {X 9.9892,Y -19.1032,Z 57,A -68.9034,B 24.8322,C -2.9881,E1 25.0758,E2 -208.5029} C_DIS
LIN {X 11.3727,Y -18.3135,Z 57,A -64.3522,B 24.831,C -2.9985,E1 25.0867,E2 -213.0648} C_DIS
LIN {X 12.4001,Y -17.634,Z 57,A -61.2117,B 24.8304,C -3.0036,E1 25.094,E2 -216.2069} C_DIS
LIN {X 13.6197,Y -16.71,Z 57,A -56.7684,B 24.8291,C -3.0157,E1 25.1038,E2 -220.6624} C_DIS
LIN {X 14.6977,Y -15.7701,Z 57,A -53.4509,B 24.8286,C -3.0197,E1 25.1106,E2 -223.9759} C_DIS
LIN {X 15.736,Y -14.7344,Z 57,A -48.7934,B 24.8267,C -3.0364,E1 25.1197,E2 -228.6529} C_DIS
LIN {X 16.8507,Y -13.4455,Z 57,A -45.0269,B 24.8262,C -3.0404,E1 25.1264,E2 -232.4116} C_DIS
LIN {X 17.5965,Y -12.4533,Z 57,A -41.5795,B 24.8251,C -3.0506,E1 25.1321,E2 -235.8666} C_DIS
LIN {X 18.2848,Y -11.4188,Z 57,A -38.5297,B 24.8243,C -3.0571,E1 25.1367,E2 -238.9166} C_DIS
LIN {X 18.9525,Y -10.2724,Z 57,A -34.7883,B 24.8229,C -3.0692,E1 25.1418,E2 -242.6673} C_DIS
LIN {X 19.7684,Y -8.5966,Z 57,A -29.0155,B 24.8202,C -3.0921,E1 25.1485,E2 -248.463} C_DIS
LIN {X 20.4129,Y -6.9298,Z 57,A -24.016,B 24.8183,C -3.109,E1 25.1531,E2 -253.4743} C_DIS
LIN {X 21.1332,Y -4.2551,Z 57,A -17.1724,B 24.8162,C -3.1262,E1 25.1575,E2 -260.3192} C_DIS
LIN {X 21.4974,Y -1.6032,Z 57,A -11.38,B 24.8152,C -3.1347,E1 25.1594,E2 -266.0974} C_DIS
LIN {X 21.5515,Y -0.4915,Z 57,A -8.3454,B 24.814,C -3.1447,E1 25.1598,E2 -269.1377} C_DIS
LIN {X 21.5433,Y 0.7736,Z 57,A -4.5424,B 24.8123,C -3.1597,E1 25.1596,E2 -272.9536} C_DIS
LIN {X 21.422,Y 2.4107,Z 57,A 0.259,B 24.8101,C -3.1777,E1 25.1583,E2 -277.769} C_DIS
LIN {X 21.2347,Y 3.7164,Z 57,A 3.6235,B 24.809,C -3.1869,E1 25.1567,E2 -281.1356} C_DIS
LIN {X 20.7029,Y 6.0082,Z 57,A 10.4244,B 24.8061,C -3.211,E1 25.1519,E2 -287.9544} C_DIS
LIN {X 19.985,Y 8.0811,Z 57,A 15.1036,B 24.8055,C -3.2159,E1 25.1474,E2 -292.6193} C_DIS
LIN {X 19.5737,Y 9.0319,Z 57,A 18.4279,B 24.8039,C -3.2292,E1 25.1435,E2 -295.957} C_DIS
LIN {X 18.7234,Y 10.6844,Z 57,A 24.1026,B 24.8014,C -3.2494,E1 25.1358,E2 -301.6501} C_DIS
LIN {X 16.8302,Y 13.4713,Z 57,A 32.2568,B 24.7997,C -3.2631,E1 25.1225,E2 -309.7973} C_DIS
LIN {X 15.8246,Y 14.6392,Z 57,A 36.4079,B 24.7985,C -3.2725,E1 25.1147,E2 -313.9524} C_DIS
LIN {X 14.4317,Y 16.0141,Z 57,A 41.5148,B 24.7974,C -3.282,E1 25.1043,E2 -319.0608} C_DIS
LIN {X 12.8718,Y 17.2927,Z 57,A 46.9963,B 24.7961,C -3.2925,E1 25.0923,E2 -324.547} C_DIS
LIN {X 11.5158,Y 18.2239,Z 57,A 51.2092,B 24.7954,C -3.2978,E1 25.0824,E2 -328.7586} C_DIS
LIN {X 10.227,Y 18.9771,Z 57,A 54.4958,B 24.7954,C -3.2973,E1 25.0744,E2 -332.0345} C_DIS
LIN {X 9.0498,Y 19.5655,Z 57,A 58.4663,B 24.7945,C -3.3054,E1 25.0644,E2 -336.0137} C_DIS
LIN {X 7.3475,Y 20.2661,Z 57,A 63.2805,B 24.794,C -3.3094,E1 25.0519,E2 -340.8268} C_DIS
LIN {X 5.8457,Y 20.7494,Z 57,A 67.2968,B 24.7938,C -3.311,E1 25.0412,E2 -344.8399} C_DIS
LIN {X 4.5106,Y 21.0797,Z 57,A 71.0608,B 24.7934,C -3.3137,E1 25.0309,E2 -348.6051} C_DIS
LIN {X 2.9632,Y 21.3528,Z 57,A 75.1768,B 24.7934,C -3.3144,E1 25.0196,E2 -352.719} C_DIS
LIN {X 1.5931,Y 21.4981,Z 57,A 78.9007,B 24.7932,C -3.3152,E1 25.0092,E2 -356.4425} C_DIS
LIN {X 0.0449,Y 21.5575,Z 57,A 83.2005,B 24.7932,C -3.3159,E1 24.9972,E2 -360.7434} C_DIS
LIN {X -1.3889,Y 21.5123,Z 57,A 86.5604,B 24.7937,C -3.3115,E1 24.9879,E2 -364.0937} C_DIS
LIN {X -2.5211,Y 21.4093,Z 57,A 90.0739,B 24.7935,C -3.3132,E1 24.9781,E2 -367.6132} C_DIS
LIN {X -4.4225,Y 21.099,Z 57,A 95.3189,B 24.7939,C -3.3101,E1 24.9637,E2 -372.8564} C_DIS
LIN {X -6.2165,Y 20.6414,Z 57,A 99.6635,B 24.7949,C -3.3016,E1 24.9521,E2 -377.1875} C_DIS
LIN {X -7.4923,Y 20.2132,Z 57,A 104.0847,B 24.7949,C -3.3022,E1 24.9404,E2 -381.619} C_DIS
LIN {X -9.8691,Y 19.1656,Z 57,A 111.3428,B 24.7959,C -3.2937,E1 24.9221,E2 -388.8754} C_DIS
LIN {X -12.0667,Y 17.8638,Z 57,A 117.0696,B 24.7981,C -3.2758,E1 24.9086,E2 -394.5772} C_DIS
LIN {X -13.0967,Y 17.1231,Z 57,A 120.4848,B 24.799,C -3.2692,E1 24.901,E2 -397.9889} C_DIS
LIN {X -14.0495,Y 16.3503,Z 57,A 123.8684,B 24.7997,C -3.2628,E1 24.8938,E2 -401.3702} C_DIS
LIN {X -15.1256,Y 15.3601,Z 57,A 127.2332,B 24.8011,C -3.2515,E1 24.8869,E2 -404.7217} C_DIS
LIN {X -15.8283,Y 14.6353,Z 57,A 130.3707,B 24.8017,C -3.2472,E1 24.8809,E2 -407.8625} C_DIS
LIN {X -16.5824,Y 13.7746,Z 57,A 133.4167,B 24.8026,C -3.2396,E1 24.8754,E2 -410.9043} C_DIS
LIN {X -17.392,Y 12.7374,Z 57,A 137.2725,B 24.8035,C -3.2322,E1 24.8689,E2 -414.7607} C_DIS
LIN {X -18.3567,Y 11.3028,Z 57,A 141.7765,B 24.8051,C -3.2193,E1 24.8621,E2 -419.2565} C_DIS
LIN {X -19.1945,Y 9.8125,Z 57,A 146.7049,B 24.8064,C -3.208,E1 24.8557,E2 -424.1842} C_DIS
LIN {X -19.8926,Y 8.3062,Z 57,A 151.4166,B 24.8079,C -3.1964,E1 24.8504,E2 -428.894} C_DIS
LIN {X -20.7512,Y 5.8392,Z 57,A 158.8961,B 24.8101,C -3.1776,E1 24.8443,E2 -436.3715} C_DIS
LIN {X -21.3602,Y 2.9101,Z 57,A 165.457,B 24.8137,C -3.1473,E1 24.841,E2 -442.8986} C_DIS
LIN {X -21.5238,Y 1.1913,Z 57,A 170.6794,B 24.8151,C -3.1355,E1 24.8399,E2 -448.1242} C_DIS
LIN {X -21.53,Y -1.0803,Z 57,A 176.7695,B 24.8173,C -3.117,E1 24.8402,E2 -454.2065} C_DIS
LIN {X -21.3448,Y -3.0176,Z 57,A -177.7645,B 24.819,C -3.1024,E1 24.842,E2 -459.6702} C_DIS
LIN {X -21.001,Y -4.8627,Z 57,A -172.3591,B 24.8206,C -3.0892,E1 24.8452,E2 -465.0759} C_DIS
LIN {X -20.1198,Y -7.74,Z 57,A -165.2965,B 24.8237,C -3.0621,E1 24.8515,E2 -472.1138} C_DIS
LIN {X -19.1143,Y -9.9682,Z 57,A -157.6665,B 24.8252,C -3.0496,E1 24.8608,E2 -479.7552} C_DIS
LIN {X -17.905,Y -12.0056,Z 57,A -152.4738,B 24.8276,C -3.0285,E1 24.8684,E2 -484.9239} C_DIS
LIN {X -17.0336,Y -13.213,Z 57,A -148.1553,B 24.8285,C -3.0209,E1 24.8757,E2 -489.245} C_DIS
LIN {X -15.7551,Y -14.7136,Z 57,A -143.2126,B 24.8299,C -3.008,E1 24.8848,E2 -494.1789} C_DIS
LIN {X -14.5574,Y -15.8997,Z 57,A -138.3026,B 24.8307,C -3.0014,E1 24.8947,E2 -499.0932} C_DIS
LIN {X -12.8976,Y -17.2734,Z 57,A -132.155,B 24.8316,C -2.9937,E1 24.9082,E2 -505.2451} C_DIS
LIN {X -11.4459,Y -18.2676,Z 57,A -128.3668,B 24.8329,C -2.9815,E1 24.9171,E2 -509.0166} C_DIS
LIN {X -10.1484,Y -19.0194,Z 57,A -123.8999,B 24.8332,C -2.9791,E1 24.928,E2 -513.4906} C_DIS
LIN {X -8.8177,Y -19.6712,Z 57,A -120.2641,B 24.8339,C -2.9729,E1 24.9372,E2 -517.1207} C_DIS
LIN {X -7.6037,Y -20.1715,Z 57,A -116.5105,B 24.8341,C -2.9713,E1 24.9469,E2 -520.8786} C_DIS
LIN {X -5.8884,Y -20.7371,Z 57,A -112.1681,B 24.8348,C -2.9649,E1 24.9585,E2 -525.2133} C_DIS
LIN {X -4.7787,Y -21.0209,Z 57,A -109.1293,B 24.835,C -2.9633,E1 24.9667,E2 -528.2525} C_DIS
LIN {X -3.7292,Y -21.2325,Z 57,A -105.9929,B 24.8349,C -2.9643,E1 24.9754,E2 -531.3946} C_DIS
LIN {X -2.3315,Y -21.4307,Z 57,A -101.7835,B 24.8346,C -2.9671,E1 24.9871,E2 -535.6134} C_DIS
LIN {X -0.0141,Y -21.5573,Z 57,A -96.0723,B 24.8348,C -2.9644,E1 25.003,E2 -541.3192} C_DIS
Enddeposition()
LIN {X -0.0141,Y -21.5573,Z 57,A -96.0723,B 24.8348,C -2.9644,E1 25.003,E2 -541.3192} C_DIS
Startdeposition()
$VEL.CP = VEL_PRINT
LIN {X -0.4329,Y -20.5645,Z 57,A -99.0748,B 24.8344,C -2.9681,E1 24.9946,E2 -538.3255} C_DIS
LIN {X -1.5637,Y -20.5094,Z 57,A -102.2317,B 24.8344,C -2.9681,E1 24.9858,E2 -535.1673} C_DIS
LIN {X -2.8546,Y -20.3697,Z 57,A -106.178,B 24.8346,C -2.9665,E1 24.9749,E2 -531.2144} C_DIS
LIN {X -4.4457,Y -20.083,Z 57,A -110.6861,B 24.8344,C -2.9682,E1 24.9625,E2 -526.7054} C_DIS
LIN {X -6.1012,Y -19.6432,Z 57,A -115.3827,B 24.834,C -2.9717,E1 24.9499,E2 -522.0095} C_DIS
LIN {X -7.6158,Y -19.1069,Z 57,A -120.0827,B 24.8337,C -2.9744,E1 24.9376,E2 -517.3061} C_DIS
LIN {X -9.4275,Y -18.2816,Z 57,A -125.5881,B 24.833,C -2.981,E1 24.9238,E2 -511.8023} C_DIS
LIN {X -10.6742,Y -17.5827,Z 57,A -130.6842,B 24.833,C -2.9809,E1 24.9116,E2 -506.6903} C_DIS
LIN {X -13.1171,Y -15.844,Z 57,A -138.8986,B 24.8313,C -2.996,E1 24.8935,E2 -498.4821} C_DIS
LIN {X -15.5482,Y -13.4666,Z 57,A -148.1007,B 24.8289,C -3.0171,E1 24.8758,E2 -489.2905} C_DIS
LIN {X -16.9381,Y -11.6699,Z 57,A -153.5379,B 24.8268,C -3.0359,E1 24.8668,E2 -483.872} C_DIS
LIN {X -17.6453,Y -10.5709,Z 57,A -157.7097,B 24.8259,C -3.0429,E1 24.8607,E2 -479.6958} C_DIS
LIN {X -18.6194,Y -8.7399,Z 57,A -162.7569,B 24.8238,C -3.0613,E1 24.8543,E2 -474.6654} C_DIS
LIN {X -19.2855,Y -7.1519,Z 57,A -169.1284,B 24.8229,C -3.0689,E1 24.8478,E2 -468.2766} C_DIS
LIN {X -20.0963,Y -4.384,Z 57,A -175.3573,B 24.8194,C -3.0991,E1 24.8433,E2 -462.0839} C_DIS
LIN {X -20.2884,Y -3.3853,Z 57,A 179.7948,B 24.8193,C -3.1006,E1 24.841,E2 -457.2107} C_DIS
LIN {X -20.5687,Y -0.2204,Z 57,A 172.1717,B 24.8155,C -3.1322,E1 24.8398,E2 -449.6174} C_DIS
LIN {X -20.5302,Y 1.2595,Z 57,A 168.6677,B 24.8138,C -3.1472,E1 24.8401,E2 -446.1283} C_DIS
LIN {X -20.4179,Y 2.4877,Z 57,A 164.7399,B 24.8127,C -3.1561,E1 24.8412,E2 -442.1985} C_DIS
LIN {X -20.1721,Y 4.0225,Z 57,A 159.8285,B 24.8113,C -3.1675,E1 24.8437,E2 -437.2852} C_DIS
LIN {X -19.8202,Y 5.4989,Z 57,A 156.157,B 24.8095,C -3.1824,E1 24.8462,E2 -433.628} C_DIS
LIN {X -19.4015,Y 6.8309,Z 57,A 151.931,B 24.8083,C -3.1929,E1 24.8499,E2 -429.4031} C_DIS
LIN {X -18.8133,Y 8.3149,Z 57,A 147.3585,B 24.8067,C -3.2056,E1 24.8549,E2 -424.8354} C_DIS
LIN {X -18.126,Y 9.7202,Z 57,A 144.1758,B 24.8047,C -3.2225,E1 24.8588,E2 -421.6762} C_DIS
LIN {X -17.5176,Y 10.7809,Z 57,A 139.2444,B 24.8043,C -3.2261,E1 24.8659,E2 -416.7278} C_DIS
LIN {X -16.6711,Y 12.0485,Z 57,A 134.5978,B 24.8031,C -3.2358,E1 24.8734,E2 -412.0817} C_DIS
LIN {X -15.1243,Y 13.9408,Z 57,A 128.4647,B 24.8007,C -3.2554,E1 24.8845,E2 -405.9678} C_DIS
LIN {X -14.014,Y 15.0565,Z 57,A 123.9534,B 24.7995,C -3.2649,E1 24.8936,E2 -401.4606} C_DIS
LIN {X -12.2699,Y 16.5082,Z 57,A 117.3053,B 24.798,C -3.2767,E1 24.9081,E2 -394.8159} C_DIS
LIN {X -10.7393,Y 17.5429,Z 57,A 112.5625,B 24.7966,C -3.288,E1 24.9192,E2 -390.085} C_DIS
LIN {X -9.5877,Y 18.1979,Z 57,A 109.2626,B 24.7956,C -3.2961,E1 24.9273,E2 -386.7949} C_DIS
LIN {X -8.1136,Y 18.901,Z 57,A 103.5049,B 24.7956,C -3.2966,E1 24.942,E2 -381.0244} C_DIS
LIN {X -5.786,Y 19.7383,Z 57,A 97.2912,B 24.7941,C -3.3081,E1 24.9584,E2 -374.827} C_DIS
LIN {X -4.4557,Y 20.0806,Z 57,A 93.9025,B 24.7934,C -3.3141,E1 24.9676,E2 -371.4479} C_DIS
LIN {X -2.9902,Y 20.3509,Z 57,A 89.1947,B 24.7934,C -3.3137,E1 24.9805,E2 -366.7347} C_DIS
LIN {X -1.0259,Y 20.5432,Z 57,A 83.2181,B 24.7934,C -3.3131,E1 24.9972,E2 -360.7543} C_DIS
LIN {X 1.2497,Y 20.5308,Z 57,A 77.3981,B 24.793,C -3.317,E1 25.0134,E2 -354.945} C_DIS
LIN {X 3.1631,Y 20.3245,Z 57,A 72.5735,B 24.7927,C -3.3196,E1 25.0267,E2 -350.1303} C_DIS
LIN {X 4.6548,Y 20.0351,Z 57,A 67.837,B 24.7934,C -3.3142,E1 25.0397,E2 -345.3868} C_DIS
LIN {X 6.3116,Y 19.5764,Z 57,A 62.8786,B 24.7939,C -3.3095,E1 25.053,E2 -340.4261} C_DIS
LIN {X 7.5334,Y 19.1397,Z 57,A 59.3483,B 24.7943,C -3.3068,E1 25.0622,E2 -336.897} C_DIS
LIN {X 9.3438,Y 18.3242,Z 57,A 53.5,B 24.7954,C -3.2979,E1 25.0769,E2 -331.0428} C_DIS
LIN {X 10.6473,Y 17.5991,Z 57,A 49.8497,B 24.7956,C -3.296,E1 25.0856,E2 -327.3993} C_DIS
LIN {X 11.8173,Y 16.8358,Z 57,A 46.3841,B 24.796,C -3.2934,E1 25.0936,E2 -323.939} C_DIS
LIN {X 12.7266,Y 16.1593,Z 57,A 43.0521,B 24.7968,C -3.2864,E1 25.101,E2 -320.6028} C_DIS
LIN {X 13.8648,Y 15.1941,Z 57,A 38.5698,B 24.7982,C -3.2757,E1 25.1104,E2 -316.1128} C_DIS
LIN {X 15.0745,Y 13.9945,Z 57,A 34.023,B 24.7992,C -3.2675,E1 25.1193,E2 -311.566} C_DIS
LIN {X 16.0204,Y 12.9011,Z 57,A 29.7641,B 24.8005,C -3.2563,E1 25.1269,E2 -307.3002} C_DIS
LIN {X 17.1599,Y 11.3398,Z 57,A 24.7559,B 24.8017,C -3.2466,E1 25.1349,E2 -302.2936} C_DIS
LIN {X 17.9942,Y 9.965,Z 57,A 20.163,B 24.8033,C -3.234,E1 25.1413,E2 -297.6943} C_DIS
LIN {X 18.7341,Y 8.4923,Z 57,A 15.613,B 24.8048,C -3.2219,E1 25.1468,E2 -293.1401} C_DIS
LIN {X 19.2829,Y 7.159,Z 57,A 11.8593,B 24.8058,C -3.2131,E1 25.1506,E2 -289.3863} C_DIS
LIN {X 19.7606,Y 5.7097,Z 57,A 7.268,B 24.8077,C -3.1974,E1 25.1544,E2 -284.784} C_DIS
LIN {X 20.1173,Y 4.2869,Z 57,A 3.6655,B 24.8086,C -3.1899,E1 25.1567,E2 -281.1845} C_DIS
LIN {X 20.3279,Y 3.1412,Z 57,A 0.3871,B 24.8099,C -3.1797,E1 25.1582,E2 -277.9012} C_DIS
LIN {X 20.4801,Y 1.9094,Z 57,A -3.0692,B 24.8111,C -3.1691,E1 25.1593,E2 -274.4402} C_DIS
LIN {X 20.5664,Y 0.3424,Z 57,A -7.9477,B 24.8134,C -3.1506,E1 25.1598,E2 -269.5469} C_DIS
LIN {X 20.511,Y -1.5411,Z 57,A -12.7543,B 24.8148,C -3.1385,E1 25.1591,E2 -264.7403} C_DIS
LIN {X 20.35,Y -2.9967,Z 57,A -16.8235,B 24.8163,C -3.1259,E1 25.1576,E2 -260.6652} C_DIS
LIN {X 20.0846,Y -4.4381,Z 57,A -20.7234,B 24.8176,C -3.1151,E1 25.1555,E2 -256.7624} C_DIS
LIN {X 19.7776,Y -5.65,Z 57,A -23.9896,B 24.8186,C -3.1065,E1 25.1531,E2 -253.4947} C_DIS
LIN {X 19.3486,Y -6.9789,Z 57,A -27.8278,B 24.8199,C -3.0953,E1 25.1497,E2 -249.6515} C_DIS
LIN {X 18.9006,Y -8.1146,Z 57,A -31.8973,B 24.8218,C -3.0787,E1 25.1454,E2 -245.5653} C_DIS
LIN {X 17.9804,Y -9.9898,Z 57,A -37.8717,B 24.8239,C -3.0606,E1 25.1376,E2 -239.5795} C_DIS
LIN {X 16.9876,Y -11.5973,Z 57,A -42.9797,B 24.8254,C -3.0477,E1 25.1298,E2 -234.4664} C_DIS
LIN {X 15.8126,Y -13.1549,Z 57,A -48.0078,B 24.8266,C -3.0374,E1 25.1211,E2 -229.4376} C_DIS
LIN {X 14.7081,Y -14.3794,Z 57,A -52.7872,B 24.828,C -3.0246,E1 25.112,E2 -224.6486} C_DIS
LIN {X 13.5864,Y -15.4435,Z 57,A -57.2793,B 24.8293,C -3.0132,E1 25.1027,E2 -220.1475} C_DIS
LIN {X 12.2094,Y -16.5537,Z 57,A -62.1008,B 24.8304,C -3.0039,E1 25.092,E2 -215.3216} C_DIS
LIN {X 10.4469,Y -17.7187,Z 57,A -67.1116,B 24.8308,C -3.0005,E1 25.0802,E2 -210.3188} C_DIS
LIN {X 9.349,Y -18.3215,Z 57,A -70.7846,B 24.8316,C -2.9931,E1 25.0711,E2 -206.6388} C_DIS
LIN {X 8.3269,Y -18.8081,Z 57,A -74.058,B 24.8323,C -2.9874,E1 25.0628,E2 -203.36} C_DIS
LIN {X 7.1781,Y -19.2757,Z 57,A -77.5148,B 24.8328,C -2.9827,E1 25.0538,E2 -199.8997} C_DIS
LIN {X 5.8761,Y -19.7118,Z 57,A -81.5017,B 24.8334,C -2.977,E1 25.0432,E2 -195.9066} C_DIS
LIN {X 4.3932,Y -20.0943,Z 57,A -85.8254,B 24.8339,C -2.9725,E1 25.0314,E2 -191.5785} C_DIS
LIN {X 3.0048,Y -20.3484,Z 57,A -89.6396,B 24.8342,C -2.9705,E1 25.0209,E2 -187.7634} C_DIS
LIN {X 1.3223,Y -20.5263,Z 57,A -94.5578,B 24.8346,C -2.9667,E1 25.0072,E2 -182.8388} C_DIS
LIN {X -0.0141,Y -20.5645,Z 57,A -97.0545,B 24.8337,C -2.9743,E1 25.0003,E2 -180.3607} C_DIS
Enddeposition()
LIN {X -0.0141,Y -20.5645,Z 57,A -97.0545,B 24.8337,C -2.9743,E1 25.0003,E2 -180.3607} C_DIS
Startdeposition()
$VEL.CP = VEL_PRINT
LIN {X 0.0281,Y -19.5811,Z 57,A -95.7793,B 24.8309,C -2.9992,E1 25.004,E2 -181.695} C_DIS
LIN {X 1.4552,Y -19.5264,Z 57,A -92.0291,B 24.8311,C -2.9979,E1 25.0145,E2 -185.4407} C_DIS
LIN {X 2.5683,Y -19.4116,Z 57,A -88.2732,B 24.8305,C -3.0033,E1 25.0249,E2 -189.2066} C_DIS
LIN {X 4.096,Y -19.1475,Z 57,A -84.6268,B 24.8308,C -3.0004,E1 25.0349,E2 -192.842} C_DIS
LIN {X 5.5591,Y -18.7749,Z 57,A -78.597,B 24.8289,C -3.0174,E1 25.0512,E2 -198.9022} C_DIS
LIN {X 7.4226,Y -18.1191,Z 57,A -74.3092,B 24.8293,C -3.0132,E1 25.0623,E2 -203.1708} C_DIS
LIN {X 8.5806,Y -17.6006,Z 57,A -69.8565,B 24.828,C -3.0248,E1 25.0736,E2 -207.6397} C_DIS
LIN {X 9.9679,Y -16.8538,Z 57,A -65.2243,B 24.8271,C -3.033,E1 25.0849,E2 -212.2775} C_DIS
LIN {X 11.5312,Y -15.8254,Z 57,A -60.1523,B 24.8263,C -3.0402,E1 25.0965,E2 -217.3494} C_DIS
LIN {X 12.6758,Y -14.9243,Z 57,A -55.2716,B 24.8246,C -3.0549,E1 25.1071,E2 -222.2461} C_DIS
LIN {X 14.3721,Y -13.2987,Z 57,A -48.2134,B 24.8225,C -3.0728,E1 25.1209,E2 -229.3169} C_DIS
LIN {X 15.8401,Y -11.511,Z 57,A -41.711,B 24.8207,C -3.088,E1 25.132,E2 -235.8243} C_DIS
LIN {X 16.8362,Y -9.9976,Z 57,A -37.3695,B 24.8201,C -3.0936,E1 25.1384,E2 -240.1573} C_DIS
LIN {X 17.4286,Y -8.9248,Z 57,A -33.2484,B 24.8183,C -3.1089,E1 25.1438,E2 -244.2928} C_DIS
LIN {X 18.0328,Y -7.6305,Z 57,A -28.8419,B 24.8166,C -3.1233,E1 25.1488,E2 -248.7095} C_DIS
LIN {X 18.7779,Y -5.5491,Z 57,A -23.2345,B 24.8153,C -3.1346,E1 25.1538,E2 -254.3119} C_DIS
LIN {X 19.0982,Y -4.3202,Z 57,A -18.6267,B 24.8129,C -3.1546,E1 25.1568,E2 -258.9406} C_DIS
LIN {X 19.4358,Y -2.3797,Z 57,A -13.489,B 24.8115,C -3.1665,E1 25.1589,E2 -264.0761} C_DIS
LIN {X 19.5488,Y -1.1184,Z 57,A -9.8119,B 24.8101,C -3.1777,E1 25.1597,E2 -267.7581} C_DIS
LIN {X 19.5798,Y 0.246,Z 57,A -5.5359,B 24.8083,C -3.1929,E1 25.1597,E2 -272.0446} C_DIS
LIN {X 19.5073,Y 1.691,Z 57,A -1.3339,B 24.8067,C -3.2057,E1 25.1588,E2 -276.252} C_DIS
LIN {X 19.2873,Y 3.3795,Z 57,A 3.5127,B 24.8051,C -3.2195,E1 25.1568,E2 -281.1029} C_DIS
LIN {X 18.9212,Y 5.0386,Z 57,A 8.3743,B 24.8034,C -3.2333,E1 25.1536,E2 -285.969} C_DIS
LIN {X 18.4207,Y 6.6389,Z 57,A 13.3297,B 24.8016,C -3.2479,E1 25.1492,E2 -290.931} C_DIS
LIN {X 17.8731,Y 7.9968,Z 57,A 17.3809,B 24.8004,C -3.2576,E1 25.1447,E2 -294.9831} C_DIS
LIN {X 17.2064,Y 9.3462,Z 57,A 21.8001,B 24.7989,C -3.2695,E1 25.139,E2 -299.407} C_DIS
LIN {X 16.7046,Y 10.2156,Z 57,A 25.5887,B 24.797,C -3.2848,E1 25.1335,E2 -303.2126} C_DIS
LIN {X 15.3132,Y 12.2034,Z 57,A 32.6579,B 24.795,C -3.3012,E1 25.1216,E2 -310.2871} C_DIS
LIN {X 13.3166,Y 14.3556,Z 57,A 40.2888,B 24.7938,C -3.3108,E1 25.1068,E2 -317.908} C_DIS
LIN {X 12.5274,Y 15.0491,Z 57,A 43.8171,B 24.7926,C -3.3203,E1 25.0992,E2 -321.4453} C_DIS
LIN {X 11.0046,Y 16.196,Z 57,A 48.6644,B 24.7922,C -3.3236,E1 25.0883,E2 -326.2834} C_DIS
LIN {X 9.8186,Y 16.9414,Z 57,A 53.143,B 24.7911,C -3.3325,E1 25.0775,E2 -330.7692} C_DIS
LIN {X 8.4653,Y 17.6561,Z 57,A 57.5484,B 24.7904,C -3.3374,E1 25.0666,E2 -335.1743} C_DIS
LIN {X 7.1999,Y 18.2091,Z 57,A 61.2883,B 24.7902,C -3.3393,E1 25.0569,E2 -338.9099} C_DIS
LIN {X 5.8996,Y 18.6704,Z 57,A 65.5882,B 24.7895,C -3.3445,E1 25.0455,E2 -343.2138} C_DIS
LIN {X 4.3275,Y 19.0966,Z 57,A 70.7126,B 24.7889,C -3.3496,E1 25.0316,E2 -348.343} C_DIS
LIN {X 2.789,Y 19.3812,Z 57,A 75.0577,B 24.7889,C -3.3494,E1 25.0197,E2 -352.6833} C_DIS
LIN {X 1.2507,Y 19.5406,Z 57,A 79.2704,B 24.7891,C -3.3477,E1 25.008,E2 -356.8896} C_DIS
LIN {X -0.0088,Y 19.5811,Z 57,A 83.298,B 24.7889,C -3.3493,E1 24.9967,E2 -360.9205} C_DIS
LIN {X -1.4428,Y 19.5273,Z 57,A 87.2053,B 24.7894,C -3.346,E1 24.9859,E2 -364.8211} C_DIS
LIN {X -2.83,Y 19.3755,Z 57,A 91.3327,B 24.7896,C -3.3439,E1 24.9744,E2 -368.9464} C_DIS
LIN {X -4.1102,Y 19.1443,Z 57,A 95.1908,B 24.79,C -3.3412,E1 24.9639,E2 -372.8024} C_DIS
LIN {X -5.3992,Y 18.8217,Z 57,A 98.987,B 24.7905,C -3.3368,E1 24.9536,E2 -376.5939} C_DIS
LIN {X -6.5601,Y 18.4491,Z 57,A 102.572,B 24.791,C -3.3327,E1 24.9442,E2 -380.1758} C_DIS
LIN {X -7.8034,Y 17.9585,Z 57,A 106.5849,B 24.7916,C -3.3279,E1 24.9338,E2 -384.1863} C_DIS
LIN {X -9.304,Y 17.2292,Z 57,A 112.1263,B 24.7922,C -3.3233,E1 24.9201,E2 -389.7318} C_DIS
LIN {X -10.9677,Y 16.221,Z 57,A 116.713,B 24.7942,C -3.3078,E1 24.9093,E2 -394.2961} C_DIS
LIN {X -11.9759,Y 15.4916,Z 57,A 121.1009,B 24.7947,C -3.3038,E1 24.8995,E2 -398.6899} C_DIS
LIN {X -13.0796,Y 14.5718,Z 57,A 125.0174,B 24.796,C -3.2934,E1 24.8912,E2 -402.5969} C_DIS
LIN {X -13.9954,Y 13.6947,Z 57,A 128.7385,B 24.797,C -3.2848,E1 24.8838,E2 -406.3131} C_DIS
LIN {X -15.0189,Y 12.5636,Z 57,A 133.7655,B 24.7981,C -3.276,E1 24.8746,E2 -411.3419} C_DIS
LIN {X -15.9589,Y 11.3458,Z 57,A 138.5224,B 24.7995,C -3.2652,E1 24.8668,E2 -416.0958} C_DIS
LIN {X -17.2727,Y 9.2236,Z 57,A 144.5934,B 24.8025,C -3.2404,E1 24.8582,E2 -422.1388} C_DIS
LIN {X -17.9139,Y 7.9054,Z 57,A 150.203,B 24.8035,C -3.2326,E1 24.8516,E2 -427.7605} C_DIS
LIN {X -18.5631,Y 6.23,Z 57,A 155.387,B 24.8054,C -3.2166,E1 24.8468,E2 -432.9355} C_DIS
LIN {X -19.1282,Y 4.1849,Z 57,A 160.7619,B 24.8081,C -3.1948,E1 24.8431,E2 -438.2894} C_DIS
LIN {X -19.3787,Y 2.8073,Z 57,A 165.4133,B 24.8094,C -3.1839,E1 24.841,E2 -442.9424} C_DIS
LIN {X -19.5444,Y 1.1867,Z 57,A 170.2424,B 24.8111,C -3.1693,E1 24.8399,E2 -447.7655} C_DIS
LIN {X -19.5767,Y -0.4082,Z 57,A 175.241,B 24.8127,C -3.1559,E1 24.8399,E2 -452.7621} C_DIS
LIN {X -19.417,Y -2.5257,Z 57,A -179.3286,B 24.8153,C -3.1341,E1 24.8414,E2 -458.1729} C_DIS
LIN {X -19.256,Y -3.5533,Z 57,A -176.1269,B 24.8163,C -3.1255,E1 24.8429,E2 -461.3728} C_DIS
LIN {X -19.0364,Y -4.5847,Z 57,A -172.5916,B 24.8172,C -3.1179,E1 24.8451,E2 -464.9107} C_DIS
LIN {X -18.4691,Y -6.5037,Z 57,A -166.9873,B 24.8193,C -3.1,E1 24.8499,E2 -470.5042} C_DIS
LIN {X -18.0492,Y -7.5914,Z 57,A -163.4134,B 24.8204,C -3.091,E1 24.8536,E2 -474.0767} C_DIS
LIN {X -17.3941,Y -8.991,Z 57,A -159.324,B 24.822,C -3.0772,E1 24.8586,E2 -478.155} C_DIS
LIN {X -16.9253,Y -9.8466,Z 57,A -155.8989,B 24.8226,C -3.072,E1 24.8633,E2 -481.5855} C_DIS
LIN {X -15.9683,Y -11.3326,Z 57,A -150.6024,B 24.824,C -3.0598,E1 24.8716,E2 -486.8792} C_DIS
LIN {X -14.7578,Y -12.8693,Z 57,A -145.2275,B 24.8257,C -3.0453,E1 24.8811,E2 -492.2444} C_DIS
LIN {X -13.9884,Y -13.7015,Z 57,A -141.1286,B 24.8261,C -3.0419,E1 24.8891,E2 -496.3528} C_DIS
LIN {X -12.4099,Y -15.1463,Z 57,A -135.2169,B 24.8276,C -3.0286,E1 24.9015,E2 -502.2558} C_DIS
LIN {X -10.9333,Y -16.2438,Z 57,A -130.435,B 24.8289,C -3.0168,E1 24.9124,E2 -507.0263} C_DIS
LIN {X -10.0542,Y -16.8028,Z 57,A -127.0565,B 24.8292,C -3.0141,E1 24.9204,E2 -510.4088} C_DIS
LIN {X -8.8727,Y -17.4551,Z 57,A -122.9119,B 24.8297,C -3.0102,E1 24.9306,E2 -514.5555} C_DIS
LIN {X -7.283,Y -18.1757,Z 57,A -117.2263,B 24.8299,C -3.0083,E1 24.9453,E2 -520.2497} C_DIS
LIN {X -4.981,Y -18.9359,Z 57,A -110.585,B 24.8308,C -3.0008,E1 24.963,E2 -526.8843} C_DIS
LIN {X -3.1842,Y -19.3202,Z 57,A -104.6678,B 24.8306,C -3.0023,E1 24.9793,E2 -532.8114} C_DIS
LIN {X -0.899,Y -19.5598,Z 57,A -98.4291,B 24.831,C -2.999,E1 24.9966,E2 -539.0448} C_DIS
LIN {X -0.899,Y -19.5598,Z 57,A -98.4291,B 24.831,C -2.999,E1 24.9966,E2 -539.0448} C_DIS
Enddeposition()
LIN {X 0.0002,Y -18.5911,Z 57,A -97.6121,B 24.8303,C -3.0047,E1 24.999,E2 -539.8753} C_DIS
Startdeposition()
$VEL.CP = VEL_PRINT
LIN {X -1.0242,Y -18.5639,Z 57,A -101.2023,B 24.8307,C -3.0017,E1 24.9889,E2 -536.2772} C_DIS
LIN {X -2.2011,Y -18.4618,Z 57,A -105.1459,B 24.8308,C -3.0002,E1 24.9779,E2 -532.3279} C_DIS
LIN {X -3.7788,Y -18.2046,Z 57,A -109.9664,B 24.8306,C -3.0025,E1 24.9647,E2 -527.5078} C_DIS
LIN {X -5.2392,Y -17.8388,Z 57,A -114.4497,B 24.8302,C -3.0061,E1 24.9526,E2 -523.0262} C_DIS
LIN {X -6.5364,Y -17.4055,Z 57,A -118.7653,B 24.8298,C -3.009,E1 24.9413,E2 -518.7092} C_DIS
LIN {X -7.8146,Y -16.8704,Z 57,A -123.2105,B 24.8294,C -3.0127,E1 24.9299,E2 -514.262} C_DIS
LIN {X -9.2835,Y -16.1089,Z 57,A -127.8657,B 24.8284,C -3.0213,E1 24.9185,E2 -509.6142} C_DIS
LIN {X -10.4468,Y -15.3803,Z 57,A -132.8219,B 24.8281,C -3.0244,E1 24.9069,E2 -504.6495} C_DIS
LIN {X -11.4433,Y -14.6542,Z 57,A -136.2905,B 24.8272,C -3.0323,E1 24.8992,E2 -501.1871} C_DIS
LIN {X -12.6745,Y -13.6031,Z 57,A -141.063,B 24.826,C -3.0427,E1 24.8892,E2 -496.4205} C_DIS
LIN {X -13.5768,Y -12.7026,Z 57,A -145.2526,B 24.8252,C -3.0498,E1 24.8811,E2 -492.2299} C_DIS
LIN {X -14.6657,Y -11.4285,Z 57,A -150.5716,B 24.8239,C -3.0609,E1 24.8717,E2 -486.9129} C_DIS
LIN {X -15.7302,Y -9.9122,Z 57,A -156.3885,B 24.8223,C -3.0746,E1 24.8626,E2 -481.0997} C_DIS
LIN {X -16.3563,Y -8.8406,Z 57,A -160.4038,B 24.8212,C -3.084,E1 24.8572,E2 -477.0857} C_DIS
LIN {X -17.1138,Y -7.2666,Z 57,A -165.5346,B 24.8194,C -3.0996,E1 24.8513,E2 -471.9642} C_DIS
LIN {X -17.6906,Y -5.7203,Z 57,A -170.4045,B 24.8176,C -3.1148,E1 24.8468,E2 -467.1031} C_DIS
LIN {X -17.9654,Y -4.7874,Z 57,A -173.7486,B 24.8167,C -3.1226,E1 24.8443,E2 -463.7582} C_DIS
LIN {X -18.3107,Y -3.2266,Z 57,A -178.6557,B 24.8149,C -3.1374,E1 24.8417,E2 -458.8577} C_DIS
LIN {X -18.5193,Y -1.6401,Z 57,A 176.8641,B 24.813,C -3.1538,E1 24.8402,E2 -454.39} C_DIS
LIN {X -18.583,Y -0.5963,Z 57,A 173.1495,B 24.8119,C -3.1624,E1 24.8398,E2 -450.6735} C_DIS
LIN {X -18.5732,Y 0.8467,Z 57,A 168.9553,B 24.8102,C -3.1769,E1 24.8401,E2 -446.489} C_DIS
LIN {X -18.4533,Y 2.2694,Z 57,A 163.7225,B 24.8088,C -3.1883,E1 24.8416,E2 -441.252} C_DIS
LIN {X -17.9495,Y 4.8469,Z 57,A 155.2541,B 24.8059,C -3.2121,E1 24.8469,E2 -432.7911} C_DIS
LIN {X -17.4473,Y 6.4237,Z 57,A 150.2974,B 24.804,C -3.2278,E1 24.8515,E2 -427.8439} C_DIS
LIN {X -16.537,Y 8.4978,Z 57,A 144.2308,B 24.8012,C -3.2508,E1 24.8587,E2 -421.7992} C_DIS
LIN {X -15.9736,Y 9.5147,Z 57,A 140.4737,B 24.8001,C -3.2602,E1 24.8639,E2 -418.0452} C_DIS
LIN {X -15.2457,Y 10.6423,Z 57,A 136.5703,B 24.7986,C -3.2721,E1 24.8699,E2 -414.1507} C_DIS
LIN {X -14.6599,Y 11.4361,Z 57,A 133.0828,B 24.7978,C -3.2785,E1 24.8758,E2 -410.6619} C_DIS
LIN {X -13.7164,Y 12.5519,Z 57,A 128.4439,B 24.7965,C -3.2891,E1 24.8844,E2 -406.0276} C_DIS
LIN {X -12.4761,Y 13.7851,Z 57,A 123.211,B 24.7949,C -3.302,E1 24.8949,E2 -400.8039} C_DIS
LIN {X -11.2335,Y 14.8156,Z 57,A 117.912,B 24.7937,C -3.3111,E1 24.9065,E2 -395.5071} C_DIS
LIN {X -9.9186,Y 15.7261,Z 57,A 113.2314,B 24.7925,C -3.3213,E1 24.9174,E2 -390.8356} C_DIS
LIN {X -8.6797,Y 16.4418,Z 57,A 109.1621,B 24.7913,C -3.3302,E1 24.9273,E2 -386.7757} C_DIS
LIN {X -7.6921,Y 16.9269,Z 57,A 105.8722,B 24.7906,C -3.3357,E1 24.9356,E2 -383.4906} C_DIS
LIN {X -6.2583,Y 17.5074,Z 57,A 100.0361,B 24.7905,C -3.3369,E1 24.9508,E2 -377.6452} C_DIS
LIN {X -4.6189,Y 18.0095,Z 57,A 95.1014,B 24.7896,C -3.344,E1 24.9641,E2 -372.7196} C_DIS
LIN {X -3.2506,Y 18.3063,Z 57,A 90.9513,B 24.7891,C -3.3482,E1 24.9754,E2 -368.575} C_DIS
LIN {X -1.4154,Y 18.5382,Z 57,A 85.2273,B 24.7887,C -3.351,E1 24.9913,E2 -362.8544} C_DIS
LIN {X 0.1484,Y 18.592,Z 57,A 80.1441,B 24.7887,C -3.3507,E1 25.0055,E2 -357.7701} C_DIS
LIN {X 1.8918,Y 18.4961,Z 57,A 74.8415,B 24.7887,C -3.3508,E1 25.0203,E2 -352.4706} C_DIS
LIN {X 3.5671,Y 18.2473,Z 57,A 69.9836,B 24.7887,C -3.3514,E1 25.0336,E2 -347.619} C_DIS
LIN {X 4.8433,Y 17.9505,Z 57,A 66.076,B 24.7889,C -3.3499,E1 25.0442,E2 -343.7139} C_DIS
LIN {X 6.1703,Y 17.5369,Z 57,A 61.9524,B 24.7891,C -3.3477,E1 25.0551,E2 -339.5927} C_DIS
LIN {X 7.2672,Y 17.1134,Z 57,A 57.7773,B 24.7901,C -3.3403,E1 25.066,E2 -335.4095} C_DIS
LIN {X 8.5444,Y 16.5133,Z 57,A 53.6085,B 24.7906,C -3.3363,E1 25.0764,E2 -331.2424} C_DIS
LIN {X 10.0385,Y 15.6498,Z 57,A 48.2823,B 24.7915,C -3.3286,E1 25.0891,E2 -325.9145} C_DIS
LIN {X 11.0487,Y 14.9538,Z 57,A 44.7983,B 24.792,C -3.3246,E1 25.097,E2 -322.4332} C_DIS
LIN {X 12.1144,Y 14.1042,Z 57,A 40.064,B 24.7935,C -3.3128,E1 25.1072,E2 -317.6889} C_DIS
LIN {X 13.4675,Y 12.8187,Z 57,A 34.2946,B 24.795,C -3.3008,E1 25.1186,E2 -311.9155} C_DIS
LIN {X 14.6054,Y 11.5052,Z 57,A 29.4678,B 24.796,C -3.293,E1 25.1272,E2 -307.0924} C_DIS
LIN {X 15.3522,Y 10.4878,Z 57,A 25.1871,B 24.7976,C -3.2803,E1 25.1341,E2 -302.8024} C_DIS
LIN {X 16.2603,Y 9.0162,Z 57,A 20.3549,B 24.7988,C -3.2709,E1 25.141,E2 -297.9726} C_DIS
LIN {X 16.8927,Y 7.7657,Z 57,A 15.8723,B 24.8004,C -3.2577,E1 25.1464,E2 -293.4829} C_DIS
LIN {X 17.5009,Y 6.2759,Z 57,A 10.1885,B 24.8029,C -3.2373,E1 25.1521,E2 -287.7823} C_DIS
LIN {X 18.175,Y 3.9155,Z 57,A 3.2098,B 24.805,C -3.2202,E1 25.1569,E2 -280.8032} C_DIS
LIN {X 18.4687,Y 2.1383,Z 57,A -2.8806,B 24.8076,C -3.1984,E1 25.1592,E2 -274.6971} C_DIS
LIN {X 18.5933,Y -0.1468,Z 57,A -9.3648,B 24.8096,C -3.1816,E1 25.1597,E2 -268.2117} C_DIS
LIN {X 18.4963,Y -1.8867,Z 57,A -14.1168,B 24.811,C -3.1705,E1 25.1587,E2 -263.4617} C_DIS
LIN {X 18.3629,Y -2.915,Z 57,A -17.8089,B 24.8127,C -3.156,E1 25.1572,E2 -259.7569} C_DIS
LIN {X 18.0969,Y -4.2647,Z 57,A -21.6046,B 24.8138,C -3.147,E1 25.155,E2 -255.9619} C_DIS
LIN {X 17.7218,Y -5.6209,Z 57,A -26.4634,B 24.8159,C -3.1291,E1 25.1511,E2 -251.0884} C_DIS
LIN {X 17.0375,Y -7.4433,Z 57,A -31.6705,B 24.8172,C -3.1184,E1 25.1457,E2 -245.8847} C_DIS
LIN {X 16.3489,Y -8.8543,Z 57,A -37.3148,B 24.8196,C -3.0973,E1 25.1385,E2 -240.2204} C_DIS
LIN {X 15.45,Y -10.3433,Z 57,A -42.4006,B 24.8211,C -3.085,E1 25.1309,E2 -235.1311} C_DIS
LIN {X 14.552,Y -11.5704,Z 57,A -45.7885,B 24.8211,C -3.084,E1 25.1253,E2 -231.757} C_DIS
LIN {X 14.0097,Y -12.2236,Z 57,A -49.3332,B 24.8229,C -3.0694,E1 25.1188,E2 -228.1938} C_DIS
LIN {X 13.29,Y -13.0024,Z 57,A -52.4558,B 24.8237,C -3.0627,E1 25.1128,E2 -225.0691} C_DIS
LIN {X 12.4308,Y -13.8261,Z 57,A -56.0368,B 24.8245,C -3.0551,E1 25.1055,E2 -221.4845} C_DIS
LIN {X 11.2825,Y -14.7783,Z 57,A -60.7582,B 24.8258,C -3.0443,E1 25.0952,E2 -216.7552} C_DIS
LIN {X 10.1985,Y -15.5461,Z 57,A -65.3893,B 24.8272,C -3.0321,E1 25.0845,E2 -212.1108} C_DIS
LIN {X 8.6534,Y -16.4561,Z 57,A -70.7899,B 24.8282,C -3.0236,E1 25.0713,E2 -206.7059} C_DIS
LIN {X 6.997,Y -17.2254,Z 57,A -76.3057,B 24.829,C -3.0162,E1 25.0572,E2 -201.1861} C_DIS
LIN {X 5.1422,Y -17.8673,Z 57,A -82.9358,B 24.8303,C -3.0051,E1 25.0395,E2 -194.5416} C_DIS
LIN {X 3.7653,Y -18.2074,Z 57,A -87.1163,B 24.8305,C -3.0026,E1 25.0281,E2 -190.3606} C_DIS
LIN {X 1.8636,Y -18.499,Z 57,A -92.6584,B 24.8307,C -3.0015,E1 25.0127,E2 -184.8202} C_DIS
LIN {X 0.4466,Y -18.5873,Z 57,A -96.6351,B 24.8306,C -3.0024,E1 25.0017,E2 -180.847} C_DIS
LIN {X 0.4466,Y -18.5873,Z 57,A -96.6351,B 24.8306,C -3.0024,E1 25.0017,E2 -180.847} C_DIS
Enddeposition()
LIN {X -0.0079,Y -17.5993,Z 57,A -96.7088,B 24.8277,C -3.0276,E1 25.0017,E2 -180.8331} C_DIS
Startdeposition()
$VEL.CP = VEL_PRINT
LIN {X 1.4555,Y -17.5438,Z 57,A -91.1712,B 24.8269,C -3.0343,E1 25.0171,E2 -186.3845} C_DIS
LIN {X 2.7228,Y -17.3925,Z 57,A -87.1045,B 24.8267,C -3.0364,E1 25.0283,E2 -190.4528} C_DIS
LIN {X 4.1555,Y -17.1067,Z 57,A -82.4316,B 24.8263,C -3.0401,E1 25.0411,E2 -195.1283} C_DIS
LIN {X 5.4739,Y -16.7313,Z 57,A -77.661,B 24.8254,C -3.0474,E1 25.0538,E2 -199.9076} C_DIS
LIN {X 7.2018,Y -16.0636,Z 57,A -71.8361,B 24.8246,C -3.0543,E1 25.0689,E2 -205.7355} C_DIS
LIN {X 8.7221,Y -15.292,Z 57,A -66.0247,B 24.8233,C -3.0656,E1 25.0832,E2 -211.557} C_DIS
LIN {X 9.7898,Y -14.6313,Z 57,A -62.5376,B 24.823,C -3.0686,E1 25.0913,E2 -215.0398} C_DIS
LIN {X 10.9265,Y -13.8031,Z 57,A -58.0159,B 24.8219,C -3.0776,E1 25.1014,E2 -219.5664} C_DIS
LIN {X 12.0326,Y -12.8504,Z 57,A -53.3605,B 24.8208,C -3.0874,E1 25.1111,E2 -224.2267} C_DIS
LIN {X 13.0102,Y -11.8596,Z 57,A -48.1768,B 24.8189,C -3.1038,E1 25.1211,E2 -229.4267} C_DIS
LIN {X 13.8265,Y -10.8969,Z 57,A -43.5678,B 24.8171,C -3.1187,E1 25.1291,E2 -234.0493} C_DIS
LIN {X 15.1159,Y -9.0238,Z 57,A -37.3675,B 24.816,C -3.1284,E1 25.1386,E2 -240.2418} C_DIS
LIN {X 15.6531,Y -8.0555,Z 57,A -33.4415,B 24.8144,C -3.1415,E1 25.1437,E2 -244.1782} C_DIS
LIN {X 16.2715,Y -6.7187,Z 57,A -28.4876,B 24.8126,C -3.157,E1 25.1492,E2 -249.1418} C_DIS
LIN {X 16.8806,Y -4.9947,Z 57,A -23.1981,B 24.8111,C -3.1691,E1 25.1539,E2 -254.43} C_DIS
LIN {X 17.2891,Y -3.3166,Z 57,A -17.5191,B 24.809,C -3.1869,E1 25.1574,E2 -260.1183} C_DIS
LIN {X 17.4833,Y -2.0606,Z 57,A -13.2846,B 24.8073,C -3.2007,E1 25.159,E2 -264.3604} C_DIS
LIN {X 17.5859,Y -0.8045,Z 57,A -9.3077,B 24.8059,C -3.2124,E1 25.1597,E2 -268.3414} C_DIS
LIN {X 17.5956,Y 0.5494,Z 57,A -4.7692,B 24.8041,C -3.2273,E1 25.1596,E2 -272.8881} C_DIS
LIN {X 17.4928,Y 1.9797,Z 57,A -0.0147,B 24.8023,C -3.2424,E1 25.1583,E2 -277.6504} C_DIS
LIN {X 17.2682,Y 3.4236,Z 57,A 4.7883,B 24.8004,C -3.2572,E1 25.156,E2 -282.4603} C_DIS
LIN {X 16.9401,Y 4.7896,Z 57,A 9.1833,B 24.799,C -3.2691,E1 25.1529,E2 -286.8584} C_DIS
LIN {X 16.4987,Y 6.1399,Z 57,A 13.746,B 24.7974,C -3.2819,E1 25.1487,E2 -291.4255} C_DIS
LIN {X 16.0305,Y 7.2757,Z 57,A 17.5469,B 24.7962,C -3.2912,E1 25.1444,E2 -295.2279} C_DIS
LIN {X 15.5516,Y 8.2501,Z 57,A 20.9189,B 24.7952,C -3.2993,E1 25.1401,E2 -298.6011} C_DIS
LIN {X 14.9289,Y 9.3297,Z 57,A 25.4359,B 24.7934,C -3.3136,E1 25.1336,E2 -303.1289} C_DIS
LIN {X 14.3232,Y 10.2353,Z 57,A 28.8146,B 24.7925,C -3.3208,E1 25.1282,E2 -306.5082} C_DIS
LIN {X 13.3714,Y 11.4507,Z 57,A 33.4506,B 24.7915,C -3.3291,E1 25.1201,E2 -311.1425} C_DIS
LIN {X 12.1921,Y 12.6992,Z 57,A 39.7423,B 24.7893,C -3.3463,E1 25.1077,E2 -317.4481} C_DIS
LIN {X 10.9034,Y 13.8212,Z 57,A 44.5954,B 24.7887,C -3.3511,E1 25.0973,E2 -322.2939} C_DIS
LIN {X 9.7118,Y 14.6832,Z 57,A 49.9421,B 24.7872,C -3.3629,E1 25.085,E2 -327.6505} C_DIS
LIN {X 8.2619,Y 15.5454,Z 57,A 55.3519,B 24.7863,C -3.3698,E1 25.0719,E2 -333.0605} C_DIS
LIN {X 6.7367,Y 16.2642,Z 57,A 61.0551,B 24.7854,C -3.3772,E1 25.0573,E2 -338.7674} C_DIS
LIN {X 5.1551,Y 16.8322,Z 57,A 66.0317,B 24.7852,C -3.3783,E1 25.0441,E2 -343.7371} C_DIS
LIN {X 3.7717,Y 17.1953,Z 57,A 70.81,B 24.7848,C -3.3816,E1 25.0312,E2 -348.5163} C_DIS
LIN {X 2.2363,Y 17.4614,Z 57,A 75.6322,B 24.7848,C -3.3815,E1 25.0179,E2 -353.3338} C_DIS
LIN {X 0.961,Y 17.5779,Z 57,A 79.9867,B 24.7847,C -3.3827,E1 25.0057,E2 -357.6891} C_DIS
LIN {X -0.4366,Y 17.599,Z 57,A 84.2321,B 24.785,C -3.3801,E1 24.9939,E2 -361.9282} C_DIS
LIN {X -1.9581,Y 17.495,Z 57,A 89.1826,B 24.7853,C -3.3778,E1 24.9801,E2 -366.8754} C_DIS
LIN {X -3.308,Y 17.2907,Z 57,A 94.7283,B 24.785,C -3.3801,E1 24.9649,E2 -372.4323} C_DIS
LIN {X -5.8329,Y 16.6096,Z 57,A 103.3099,B 24.7862,C -3.3712,E1 24.942,E2 -381.0072} C_DIS
LIN {X -7.5435,Y 15.9059,Z 57,A 109.0321,B 24.7874,C -3.3611,E1 24.9275,E2 -386.7194} C_DIS
LIN {X -9.2138,Y 15.0008,Z 57,A 115.0469,B 24.7889,C -3.3498,E1 24.9129,E2 -392.7249} C_DIS
LIN {X -10.7526,Y 13.939,Z 57,A 120.9096,B 24.7905,C -3.3369,E1 24.8997,E2 -398.5772} C_DIS
LIN {X -12.2783,Y 12.6157,Z 57,A 128.0472,B 24.7921,C -3.3242,E1 24.885,E2 -405.7133} C_DIS
LIN {X -13.3416,Y 11.4855,Z 57,A 132.2925,B 24.794,C -3.3092,E1 24.8771,E2 -409.9415} C_DIS
LIN {X -14.0871,Y 10.5578,Z 57,A 136.7597,B 24.795,C -3.3011,E1 24.8695,E2 -414.4105} C_DIS
LIN {X -15.3014,Y 8.7048,Z 57,A 144.3041,B 24.7973,C -3.2823,E1 24.8585,E2 -421.9486} C_DIS
LIN {X -16.0592,Y 7.2116,Z 57,A 149.1479,B 24.7995,C -3.2648,E1 24.8527,E2 -426.7766} C_DIS
LIN {X -16.5497,Y 6.001,Z 57,A 153.5188,B 24.801,C -3.2525,E1 24.8483,E2 -431.1426} C_DIS
LIN {X -16.9355,Y 4.8057,Z 57,A 157.7264,B 24.8025,C -3.2404,E1 24.8449,E2 -435.3455} C_DIS
LIN {X -17.3027,Y 3.246,Z 57,A 162.6137,B 24.8046,C -3.2235,E1 24.8421,E2 -440.221} C_DIS
LIN {X -17.5089,Y 1.8273,Z 57,A 167.3559,B 24.8063,C -3.2092,E1 24.8404,E2 -444.9573} C_DIS
LIN {X -17.6002,Y 0.3684,Z 57,A 172.9876,B 24.8078,C -3.1968,E1 24.8398,E2 -450.5931} C_DIS
LIN {X -17.5559,Y -1.2992,Z 57,A 178.0799,B 24.8099,C -3.1791,E1 24.8406,E2 -455.6736} C_DIS
LIN {X -17.364,Y -2.8995,Z 57,A -176.8586,B 24.8119,C -3.1626,E1 24.8426,E2 -460.7258} C_DIS
LIN {X -17.0539,Y -4.3667,Z 57,A -172.1687,B 24.8137,C -3.1475,E1 24.8455,E2 -465.4071} C_DIS
LIN {X -16.5237,Y -6.0708,Z 57,A -165.7745,B 24.8155,C -3.1325,E1 24.8512,E2 -471.8019} C_DIS
LIN {X -15.8705,Y -7.618,Z 57,A -160.3393,B 24.8173,C -3.1174,E1 24.8574,E2 -477.2307} C_DIS
LIN {X -15.3517,Y -8.6164,Z 57,A -156.6232,B 24.8184,C -3.108,E1 24.8624,E2 -480.9438} C_DIS
LIN {X -14.4286,Y -10.0864,Z 57,A -150.9379,B 24.82,C -3.0942,E1 24.8712,E2 -486.6244} C_DIS
LIN {X -13.4819,Y -11.3206,Z 57,A -146.3167,B 24.8215,C -3.081,E1 24.8792,E2 -491.2358} C_DIS
LIN {X -12.5613,Y -12.3341,Z 57,A -141.9825,B 24.8227,C -3.0712,E1 24.8875,E2 -495.5653} C_DIS
LIN {X -11.7743,Y -13.0876,Z 57,A -138.6124,B 24.8236,C -3.0635,E1 24.8944,E2 -498.9309} C_DIS
LIN {X -10.9942,Y -13.7497,Z 57,A -134.5324,B 24.8239,C -3.0606,E1 24.9032,E2 -503.0193} C_DIS
LIN {X -9.8393,Y -14.5981,Z 57,A -130.3121,B 24.825,C -3.0512,E1 24.9128,E2 -507.2317} C_DIS
LIN {X -8.7618,Y -15.2691,Z 57,A -125.6603,B 24.8254,C -3.0478,E1 24.924,E2 -511.8894} C_DIS
LIN {X -7.4801,Y -15.9363,Z 57,A -121.0515,B 24.8261,C -3.0418,E1 24.9356,E2 -516.496} C_DIS
LIN {X -6.1217,Y -16.5055,Z 57,A -116.4796,B 24.8267,C -3.0363,E1 24.9474,E2 -521.0645} C_DIS
LIN {X -4.9793,Y -16.8853,Z 57,A -112.6606,B 24.8271,C -3.033,E1 24.9576,E2 -524.8824} C_DIS
LIN {X -3.9382,Y -17.1581,Z 57,A -109.3183,B 24.8274,C -3.0303,E1 24.9667,E2 -528.2229} C_DIS
LIN {X -2.9038,Y -17.3633,Z 57,A -105.8626,B 24.8275,C -3.0292,E1 24.9762,E2 -531.6798} C_DIS
LIN {X -1.5123,Y -17.5389,Z 57,A -100.4699,B 24.827,C -3.0336,E1 24.9912,E2 -537.086} C_DIS
Enddeposition()
END
